# B&R Automation Studio project 8238 (part 29)

#### BIN_TO_BCD_INT.ab
```automation-basic
FUNCTION_BLOCK BIN_TO_BCD_INT

		(* Implementation of BIN_TO_BCD *)

	RegisterOUT = 0

		remain = RegisterIN

;		f = remain / 100000
;		remain = remain - (f * 100000)
;		e = remain / 10000
;		remain = remain - (e * 10000)
		d = remain / 1000
		remain = remain - (d * 1000)
		c = remain / 100
		remain = remain - (c * 100)
		b = remain / 10
		a = remain - (b * 10)
		RegisterOUT = RegisterIN + (b * 6) + (c * 156) + (d * 3096)// + (e * 55536)// + (f * 948576)

END_FUNCTION_BLOCK
```

#### Get_Lower2Bytes.st
```iecst
(* Copy the lower 2 bytes from a byte register *)
FUNCTION Get_Lower2Bytes

	memcpy(ADR(Get_Lower2Bytes),ADR(input),2);

END_FUNCTION
```

#### Get_Higher2Bytes.st
```iecst
(* Copy the upper 2 bytes of a DWORD to a WORD *)
FUNCTION Get_Higher2Bytes
	memcpy(ADR(Get_Higher2Bytes),ADR(input) + 2,2);
END_FUNCTION
```

#### GetPowerlinkNodeIP.st
```iecst
(* *Function to build BR camera image URL from EPL IP and Node address *)
FUNCTION_BLOCK GetPowerlinkNodeIP

	IF EDGEPOS(Enable)AND (state = 0) THEN
		state := 1;
	ELSIF (((state = 4) OR (state = 100)) AND NOT Enable) THEN
		state := 0;
	END_IF;

	getEPL_IP.enable 	:= (state = 2);

	CASE state OF
		0:  // WAIT
			Status := ERR_FUB_ENABLE_FALSE;

		1: // Build and check the interface path
			Status := ERR_FUB_BUSY;
			IF (RIGHT(EplInterfacePath,4) = '.ETH') THEN
				device := EplInterfacePath;
				state := 2;
			ELSE
				device := CONCAT(EplInterfacePath,'.ETH');
				state := 2;
			END_IF;

		2:// Get the IP address of the interface..
			Status := ERR_FUB_BUSY;
			getEPL_IP.pIPAddr 	:= ADR(eplAddress);
			getEPL_IP.Len 		:= SIZEOF(eplAddress);
			getEPL_IP.pDevice 	:= ADR(device);
			IF (getEPL_IP.status = ERR_OK) THEN
				state := 3;
				//brsstrcpy(pIPAddress,ADR(''));
			ELSIF (getEPL_IP.status <> ERR_FUB_BUSY) AND (getEPL_IP.status <> ERR_FUB_ENABLE_FALSE)  THEN
				Status := getEPL_IP.status;
				state := 100;
			END_IF;

		3://Replace the
			Status := ERR_FUB_BUSY;
			ethInetAton(ADR(eplAddress),ADR(eplIP));
			eplIP := (eplIP AND 16#00FF_FFFF) OR (16#FF00_0000 AND SHL(Node,24));// Replace the end of the IP with the node
			ethInetNtoa(eplIP,pIPAddress);
			state := 4;

		4:// Complete
			Status := ERR_OK;

		100:// Error step

	END_CASE;

	getEPL_IP();

END_FUNCTION_BLOCK
```

#### DByte_TO_4Byte.st
```iecst
(* Build 32 bit register from 2 16bit register *)
FUNCTION DByte_TO_4Byte
	memcpy(ADR(internalValue),adrLower,2);
	memcpy(ADR(internalValue)+2,adrHigher,2);
	DByte_TO_4Byte := internalValue;
END_FUNCTION
```

#### getNodeFromPV.st
```iecst
(* Get Node and Connection string from a PV var. *)
FUNCTION_BLOCK getNodeFromPV

	IF NOT enable THEN
		state := 0;
	END_IF;

	IF (state = 0) THEN // Not ENABLED
		IF enable THEN
			state := 1;
			pointer := 0;
			IF_Adr := '';
			NodeNumber := 0;
			brsmemset(ADR(searchString),0,SIZEOF(searchString));
		ELSE
			status := ERR_FUB_ENABLE_FALSE;
		END_IF;
	END_IF;

	IF (state = 1) THEN // get pointer to iom file so we can interate through the string.
		searchLen := LEN(pvName);
		mO_info(enable := (searchLen > 0), pName := ADR('iomap'), grp := 0);
		IF ((searchLen = 0) OR (searchLen > SIZEOF(searchString))) THEN
			state := 100;
			status := 101;
		ELSIF (mO_info.status = ERR_OK) THEN
			state := state := 2;
		ELSIF (mO_info.status <> ERR_FUB_BUSY) THEN
			status := mO_info.status;
			state := 100;
		END_IF;
	END_IF;

	//iterate through the string until we find our var name
	scanCount := 0;
	WHILE ((pointer < (mO_info.size - searchLen)) AND (scanCount <= 50000) AND (state = 2)) DO
		scanCount := scanCount + 1;
		brsmemcpy(ADR(searchString),(mO_info.address + pointer),searchLen);
		IF (searchString = pvName) THEN
			brsmemset(ADR(searchString),0,SIZEOF(searchString));
			state := 3;
		END_IF;
		pointer := pointer + 1;
		IF (pointer = (mO_info.size - searchLen)) THEN
			state := 20; // NOT FOUND
		END_IF;
	END_WHILE;

	// Iterate back through the string to find the start of the node
	scanCount := 0;
	WHILE ((pointer > 0) AND (pointer < (mO_info.size - searchLen)) AND (scanCount <= 250) AND (state = 3)) DO
		scanCount := scanCount + 1;
		pointer := pointer - 1;
		brsmemcpy(ADR(searchString),(mO_info.address + pointer),2);
		IF (searchString = 'ST') THEN
			startNode := pointer + 2;
			brsmemset(ADR(searchString),0,SIZEOF(searchString));
			state := 4;
		END_IF;
		IF (pointer = 0) OR (scanCount = 250) THEN
			state := 100; // ERROR;
			status := 103;
		END_IF;
	END_WHILE;

	// Iterate back through the string to find the start of the path
	scanCount := 0;
	WHILE ((pointer > 0) AND (pointer < (mO_info.size - searchLen)) AND (scanCount <= 250) AND (state = 4)) DO
		scanCount := scanCount + 1;
		pointer := pointer - 1;
		brsmemcpy(ADR(searchString),(mO_info.address + pointer),2);
		IF (searchString = '="') THEN
			startPath := pointer + 2;
			pointer := startNode;
			brsmemset(ADR(searchString),0,SIZEOF(searchString));
			state := 5;
		END_IF;
		IF (pointer = 0) OR (scanCount = 250) THEN
			state := 100; // ERROR;
			status := 104;
		END_IF;
	END_WHILE;

	// Iterate back through the string to find the end of the node
	scanCount := 0;
	WHILE ((pointer > 0) AND (pointer < (mO_info.size - 1)) AND (scanCount <= 250) AND (state = 5)) DO
		scanCount := scanCount + 1;
		pointer := pointer + 1;
		brsmemcpy(ADR(searchString),(mO_info.address + pointer),1);
		IF (searchString = '"') OR (searchString = '.') THEN
			endNode := pointer;
			state := 6;
		END_IF;
		IF (pointer = 0) OR (pointer = (mO_info.size - 1)) OR (scanCount = 250) THEN
			state := 100; // ERROR;
			status := 105;
		END_IF;
	END_WHILE;

	IF (state = 6) THEN
		brsmemset(ADR(IF_Adr),0,SIZEOF(IF_Adr));
		brsmemcpy(ADR(IF_Adr),mO_info.address + startPath, startNode - 3 - startPath);
		IF (LEFT(IF_Adr,1) = '%') THEN
			 IF_Adr := RIGHT(IF_Adr,(LEN(IF_Adr) - 4));
		END_IF;
		// Get the Node
		brsmemset(ADR(nodeString),0,SIZEOF(nodeString));
		brsmemcpy(ADR(nodeString),mO_info.address + startNode, endNode - startNode);
		NodeNumber := DINT_TO_USINT(atoi(ADR(nodeString)));
		state := 10;
	END_IF;

	IF (state = 10) THEN// Complete

	END_IF;

	IF (state = 20) THEN // NOT FOUND

	END_IF;

	IF (state = 100) THEN // ERROR
		state := 0;
	END_IF;

	IF (state = 10) THEN
		status := ERR_OK;
		state := 0;
	ELSIF (state = 20) THEN // NOT FOUND
		status := 200; // NOT FOUND
		state := 0;
	ELSIF (state > 0) AND (state < 100) THEN
		status := ERR_FUB_BUSY;
	END_IF;

END_FUNCTION_BLOCK
```

#### GetModuleName.st
```iecst
(* TODO: Add your comment here *)
FUNCTION_BLOCK GetModuleName

	IF NOT enable THEN
		state := 0;
	END_IF;

	IF (state = 0) THEN // Not ENABLED
		IF enable THEN
			state := 1;
			pointer := 0;
		ELSE
			status := ERR_FUB_ENABLE_FALSE;
		END_IF;
	END_IF;

	IF (state = 1) THEN // get pointer to iom file so we can interate through the string.
		brsstrcpy(ADR(moduleAddress),ADR('"'));
		brsstrcat(ADR(moduleAddress),pModuleAddress);
		brsstrcat(ADR(moduleAddress),ADR('"'));
		brsmemset(ADR(searchString),0,SIZEOF(searchString));
		brsmemset(ADR(ModuleName),0,SIZEOF(ModuleName));
		searchLen := LEN(moduleAddress);
		mO_info(enable := (searchLen > 0), pName := ADR('arconfig'), grp := 0);
		IF ((searchLen <= 2) OR (searchLen > SIZEOF(searchString))) THEN
			state := 100;
			status := 101;
		ELSIF (mO_info.status = ERR_OK) THEN
			state := state := 2;
		ELSIF (mO_info.status <> ERR_FUB_BUSY) THEN
			status := mO_info.status;
			state := 100;
		END_IF;
	END_IF;

	//iterate through the string until we find our address
	scanCount := 0;
	WHILE ((pointer < (mO_info.size - searchLen)) AND (scanCount <= 50000) AND (state = 2)) DO
		scanCount := scanCount + 1;
		brsmemcpy(ADR(searchString),(mO_info.address + pointer),searchLen);
		IF (searchString = moduleAddress) THEN
			brsmemset(ADR(searchString),0,SIZEOF(searchString));
			foundCount := foundCount + 1;
			state := 3;
		END_IF;
		pointer := pointer + 1;
		IF (pointer = (mO_info.size - searchLen)) THEN
			state := 20; // NOT FOUND
		END_IF;
	END_WHILE;

	// Iterate back through the string to find the module Name
	scanCount := 0;
	WHILE ((pointer > 0) AND (pointer < (mO_info.size - 1)) AND (scanCount <= 200) AND (state = 3)) DO
		scanCount := scanCount + 1;
		pointer := pointer + 1;
		brsmemcpy(ADR(searchString),(mO_info.address + pointer),42);
		IF (searchString = '<Parameter ID="HardwareModuleName" Value="')THEN
			brsmemset(ADR(searchString),0,SIZEOF(searchString));
			pointer := pointer + 42;
			start := pointer;
			state := 4;
		END_IF;
		IF (pointer = 0) OR (pointer = (mO_info.size - 1)) OR (scanCount = 200) THEN
			state := 100; // ERROR;
			status := 103;
		END_IF;
	END_WHILE;

	// Iterate back through the string to find the module Name
	scanCount := 0;
	WHILE ((pointer > 0) AND (pointer < (mO_info.size - 1)) AND (scanCount <= 100) AND (state = 4)) DO
		scanCount := scanCount + 1;
		pointer := pointer + 1;
		brsmemcpy(ADR(searchString),(mO_info.address + pointer),1);
		IF (searchString = '"')THEN
			end := pointer;
			state := 5;
		END_IF;
		IF (pointer = 0) OR (pointer = (mO_info.size - 1)) OR (scanCount = 100) THEN
			state := 100; // ERROR;
			status := 104;
		END_IF;
	END_WHILE;

	IF (state = 5) THEN
		// Get the Name
		IF ((end - start) <= SIZEOF(ModuleName)) THEN
			brsmemset(ADR(ModuleName),0,SIZEOF(ModuleName));
			brsmemcpy(ADR(ModuleName),mO_info.address + start, end - start);
			state := 10;
		ELSE
			state := 100;
			status := 105;
		END_IF;
	END_IF;

	IF (state = 10) THEN// Complete

	END_IF;

	IF (state = 20) THEN // NOT FOUND

	END_IF;

	IF (state = 100) THEN // ERROR
		state := 0;
	END_IF;

	IF (state = 10) THEN
		status := ERR_OK;
		state := 0;
	ELSIF (state = 20) THEN // NOT FOUND
		status := 200; // NOT FOUND
		state := 0;
	ELSIF (state > 0) AND (state < 100) THEN
		status := ERR_FUB_BUSY;
	END_IF;

END_FUNCTION_BLOCK
```

#### Get_LowerByte.st
```iecst
(* Copy the lower 2 bytes from a byte register *)
FUNCTION Get_LowerByte

	memcpy(ADR(Get_LowerByte),ADR(input),1);

END_FUNCTION
```

#### Get_HigherByte.st
```iecst
(* Copy the upper 2 bytes of a DWORD to a WORD *)
FUNCTION Get_HigherByte
	memcpy(ADR(Get_HigherByte),ADR(input) + 1,1);
END_FUNCTION
```

#### SetValueByName.st
```iecst
//*Set Local variable from external task
FUNCTION SetValueByName
	SetValueByName := 0;
	IF (brsstrlen(ADR(TaskName)) > 0 )THEN
		varName := '::';
		brsstrcat(ADR(varName),ADR(TaskName));
		brsstrcat(ADR(varName),ADR(':'));
		brsstrcat(ADR(varName),ADR(VarName));
	ELSE
		brsstrcpy(ADR(varName),ADR(VarName));
	END_IF;

	IF (PV_xgetadr(ADR(varName),ADR(pVar),ADR(sVar)) = 0) THEN
		IF (SIZEOF(Value) <= sVar)THEN
			brsmemcpy(pVar,ADR(Value),SIZEOF(Value));
			SetValueByName := 1;
		ELSE
			brsmemcpy(pVar,ADR(Value),sVar);
			SetValueByName := 1;
		END_IF;
	END_IF;
END_FUNCTION
```

#### GetValueByName.st
```iecst
//*Set Local variable from external task
FUNCTION GetValueByName
	GetValueByName := 0;

	IF (brsstrlen(ADR(TaskName)) > 0 )THEN
		varName := '::';
		brsstrcat(ADR(varName),ADR(TaskName));
		brsstrcat(ADR(varName),ADR(':'));
		brsstrcat(ADR(varName),ADR(VarName));
	ELSE
		brsstrcpy(ADR(varName),ADR(VarName));
	END_IF;

	status := PV_xgetadr(ADR(varName),ADR(pVar),ADR(sVar));
	IF (status = 0) THEN
		IF (sValue >= sVar)THEN
			//Clear the value
			IF (sValue > sVar) THEN
				brsmemset(pValue,0,sValue);
			END_IF;
			brsmemcpy(pValue,pVar,sVar);
			GetValueByName := 1;
		END_IF;
	END_IF;
END_FUNCTION
```

#### LoadCell.st
```iecst
FUNCTION_BLOCK LoadCell

	IF capture_weight_bool THEN
		brsmemmove(ADR(weight_array[1]), ADR(weight_array), 1498);

		weight_array[0] := analog_weight;

		IF small_interval > 0 THEN
			small_value := 0;
			FOR i := 0 TO small_interval - 1 DO
			small_value := small_value + weight_array[i];
			END_FOR;
			udp_data.small_smoothing_value := small_smoothing_value := DINT_TO_UINT(small_value / small_interval);

		END_IF;

		IF large_interval > 0 THEN
			large_value := 0;
			FOR x := 0 TO large_interval - 1 DO
			large_value := large_value + weight_array[x];
			END_FOR;

			udp_data.large_smoothing_value := large_smoothing_value := DINT_TO_UINT(large_value / large_interval);
		END_IF;

		udp_data.capture_weight := capture_weight := analog_weight;
	END_IF;

	weight_tolerance := (((server_send_weight - tare)/100) * weight_tolerance_percent);
	empty := (analog_weight <= (tare + weight_tolerance)) AND (tare > 0);
	min_weight:= (analog_weight > server_min_weight) AND (server_min_weight > 0);
	near_weight := (analog_weight > server_near_weight) AND (server_near_weight > 0);
	bufflector_door_weight := (analog_weight > server_buffer_weight) AND (server_buffer_weight > 0);
	notify_weight := (analog_weight > server_notify_weight) AND (server_notify_weight > 0);
	full := (analog_weight > server_send_weight) AND (server_send_weight > 0);
	over_weight:= (analog_weight >= server_over_weight);

	IF span > 0 THEN
		udp_data.capture_weight_value := capture_weight_value := (((udp_data.capture_weight - tare) * 100) / span);
		udp_data.live_weight_value := live_weight_value := (((analog_weight - tare) * 100) / span);
		udp_data.small_smoothing_weight := small_smoothing_weight := (((udp_data.small_smoothing_value - tare) * 100) / span);
		udp_data.large_smoothing_weight := large_smoothing_weight := (((udp_data.large_smoothing_value - tare) * 100) / span);
	END_IF;

END_FUNCTION_BLOCK
```

#### BCD_ENCODE.st
```iecst
(* TODO: Add your comment here *)
FUNCTION_BLOCK BCD_Encode

	Output := 0;

	IF Input.0 THEN
		Output := Output + 1;
	END_IF;
	IF Input.1 THEN
		Output := Output + 2;
	END_IF;
	IF Input.2 THEN
		Output := Output + 4;
	END_IF;
	IF Input.3 THEN
		Output := Output + 8;
	END_IF;
	IF Input.4 THEN
		Output := Output + 10;
	END_IF;
	IF Input.5 THEN
		Output := Output + 20;
	END_IF;
	IF Input.6 THEN
		Output := Output + 40;
	END_IF;
	IF Input.7 THEN
		Output := Output + 80;
	END_IF;
	IF Input.8 THEN
		Output := Output + 100;
	END_IF;
	IF Input.9 THEN
		Output := Output + 200;
	END_IF;
	IF Input.10 THEN
		Output := Output + 400;
	END_IF;
	IF Input.11 THEN
		Output := Output + 800;
	END_IF;
	IF Input.12 THEN
		Output := Output + 1000;
	END_IF;
	IF Input.13 THEN
		Output := Output + 2000;
	END_IF;
	IF Input.14 THEN
		Output := Output + 4000;
	END_IF;
	IF Input.15 THEN
		Output := Output + 8000;
	END_IF;

END_FUNCTION_BLOCK
```

#### Types.typ
```iecst
TYPE
RailComm_typ :STRUCT
  Messages : RailMessages_typ;
END_STRUCT;
RailMessages_typ : STRUCT
  Write : UINT;
  Read : ARRAY[0..15] OF UINT;
END_STRUCT;
SlingInput_typ : STRUCT
  Write : UINT;
  Read : UDINT;
END_STRUCT;
  bnr_io : STRUCT
    X01 : BOOL;
    X02 : BOOL;
    X03 : BOOL;
    X04 : BOOL;
    X05 : BOOL;
    X06 : BOOL;
    X07 : BOOL;
    X08 : BOOL;
    X09 : BOOL;
    X10 : BOOL;
    X11 : BOOL;
    X12 : BOOL;
    X13 : BOOL;
    X14 : BOOL;
    X15 : BOOL;
    X16 : BOOL;
    X17 : BOOL;
    X18 : BOOL;
    X19 : BOOL;
    X20 : BOOL;
    Y01 : BOOL;
    Y02 : BOOL;
    Y03 : BOOL;
    Y04 : BOOL;
    Y05 : BOOL;
    Y06 : BOOL;
    Y07 : BOOL;
    Y08 : BOOL;
    Y09 : BOOL;
    Y10 : BOOL;
    Y11 : BOOL;
    Y12 : BOOL;
    Y13 : BOOL;
    Y14 : BOOL;
    Y15 : BOOL;
    Y16 : BOOL;
    Y17 : BOOL;
    Y18 : BOOL;
    Y19 : BOOL;
    Y20 : BOOL;
  END_STRUCT;

  rail : 	STRUCT
    ac : BOOL;
    activity : BOOL;
    after : BOOL;
    after_raw : BOOL;
    after_a : BOOL;
    after_a_raw : BOOL;
    after_b : BOOL;
    after_b_raw : BOOL;
    air_pressure : BOOL;
    alarm : BOOL;
    alarm_time : TIME;
    arm: BOOL;
    arrive : BOOL;
    arrive_raw : BOOL;
    at_rail : BOOL;
    bag_emptied : BOOL;
    before : BOOL;
    before_raw : BOOL;
    bnx : BOOL;
    bottom_door : BOOL;
    bottom_door_sensor : BOOL;
    bring_ok : BOOL;
    bufflector_door_weight : BOOL;
    buffer_protection : BOOL;
    busy : BOOL;
    cake_break_bypass : BOOL;
    cake_break_done : BOOL;
    cake_break_signal : BOOL;
    cake_break_start : BOOL;
    cake_close : BOOL;
    cake_left : BOOL;
    cake_open : BOOL;
    cake_right : BOOL;
    call_button : BOOL;
    capture_weight: BOOL;
    catch : BOOL;
    cc_open_bottom : BOOL;
    cc_open_bottom_os : BOOL;
    cc_open_top : BOOL;
    cc_open_top_os : BOOL;
    cc_shut_bottom : BOOL;
    cc_shut_bottom_os : BOOL;
    cc_shut_top : BOOL;
    cc_shut_top_os : BOOL;
    change_reset : BOOL;
    chute : BOOL;
    chute_clear : BOOL;
    chute_in_position : BOOL;
    clamp : BOOL;
    clear_belt : BOOL;
    close : BOOL;
    close_bottom : BOOL;
    close_top : BOOL;
    closed : BOOL;
    comm_ok : BOOL;
    counter : USINT;
    conv_estop : BOOL;
    conv_fwd : BOOL;
    conv_rev : BOOL;
    conveyor_running : BOOL;
    custom_bring_lock : BOOL;
    custom_send_lock : BOOL;
    cycle_count : INT;
    cylinderAtReceive : BOOL;
    cylinderAtRelease : BOOL;
    dampner : BOOL;
    dampner_closed : BOOL;
    dampner_open : BOOL;
    debagger_arm : BOOL;
    delayed_bottom_door : BOOL;
    destination : INT;
    device_received : BOOL;
    device_receive_ok : BOOL;
    device_release_ok : BOOL;
    dog_sensor : BOOL;
    done : BOOL;
    done_smashing : BOOL;
    door_sensor : BOOL;
    down : BOOL;
    down_button : BOOL;
    down_raw : BOOL;
    emergency_cut_off : BOOL;
    empty : BOOL;
    empty_bag : BOOL;
    energize : BOOL;
    fire : BOOL;
    fire_cyl_receive : BOOL;
    fire_cyl_release : BOOL;
    fire_down : BOOL;
    fire_f_trig : F_TRIG;
    fire_r_trig : R_TRIG;
    fire_ns : BOOL;
    fire_os : BOOL;
    fire_up : BOOL;
    fired: BOOL;
    firing : BOOL;
    firing_reset : BOOL;
    flip : BOOL;
    flipped : BOOL;
    fnx : BOOL;
    foot : BOOL;
    front : BOOL;
    front_a : BOOL;
    front_b : BOOL;
    front_bag_mt : BOOL;
    front_raw : BOOL;
    front_stp : BOOL;
    full : BOOL;
    full_sensor : BOOL;
    green_light : BOOL;
    going_to : BOOL;
    going_to_os : BOOL;
    going_to_ns : BOOL;
    going_to_r_trig : R_TRIG;
    going_to_f_trig : F_TRIG;
    grab : BOOL;
    high_valve : BOOL;
    input_enabled : BOOL;
    insert : BOOL;
    insert_reset : BOOL;
    in_pos : BOOL; (*In position after dbnc*)
    in_pos_raw : BOOL;  (*In position sensor*)
    inx : BOOL;
    io_ok : BOOL;
    io_ok_A : BOOL;
    io_ok_B : BOOL;
    io_ok_C : BOOL;
    jogmode : BOOL;
    latch : BOOL;
    latched : BOOL;
    leave1 : BOOL;
    leave2 : BOOL;
    leave3 : BOOL;
    level_arm : BOOL;
    lift_stp : BOOL;
    LFT1 : BOOL;
    LFT1_RAW : BOOL;
    LFT2 : BOOL;
    LFT2_RAW : BOOL;
    LFT3 : BOOL;
    LFT3_RAW : BOOL;
    LFT4 : BOOL;
    LFT4_RAW : BOOL;
    LFT5 : BOOL;
    LFT5_RAW : BOOL;
    lift_clamp : BOOL;
    lift_jammed : BOOL;
    lift_position : INT;
    lift_running : BOOL;
    loaded : BOOL;
    loading_position : BOOL;
    loading_position_raw : BOOL;
    loading_signal : BOOL;
    lockout : BOOL;
    log_dist : INT;
    log_now_a : BOOL;
    log_now_b : BOOL;
    low_air_alarm : BOOL;
    low_valve : BOOL;
    man_open : BOOL;
    man_send : BOOL;
    man_send_button_1 : BOOL;
    man_send_button_2 : BOOL;
    man_send_button : BOOL;
    manual_mode : BOOL;
    marker_made : BOOL;
    mid : BOOL;
    mid_raw : BOOL;
    min_weight : BOOL;
    min_weight_send : BOOL;
    mod_count : INT;
    move_rail : BOOL;
    move_rail_up : BOOL;
    move_rail_down : BOOL;
    mt_arrived : BOOL;
    near_weight : BOOL;
    near_weight_send : BOOL;
    need_to_empty_bd : BOOL;
    need_to_empty_td : BOOL;
    next_rails_ok : BOOL;
    no_dests_ok : BOOL;
    not_io_ok : BOOL;
    notify_weight : BOOL;
    oc : BOOL;
    ok_to_send : BOOL;
    onoff : BOOL;
    open : BOOL;
    open_bottom : BOOL;
    open_manual : BOOL;
    open_signal : BOOL;
    open_pendant : BOOL;
    opened : BOOL;
    out1 : BOOL;
    over_full_sensor : BOOL;
    over_full_light : BOOL;
    over_weight : BOOL;
    paddle_sensor : BOOL;
    pilot_light : BOOL;
    poa : BOOL;
    pos1 : BOOL;
    pos1_raw : BOOL;
    pos2 : BOOL;
    pos2_raw : BOOL;
    pos3 : BOOL;
    pos3_raw : BOOL;
    pos4 : BOOL;
    pos4_raw : BOOL;
    pos_1_after_raw : BOOL;
    pos_1_after : BOOL;
    pos_2_after_raw : BOOL;
    pos_2_after : BOOL;
    pos_3_after_raw : BOOL;
    pos_3_after : BOOL;
    pos_4_after_raw : BOOL;
    pos_4_after : BOOL;
    pos_5_after_raw : BOOL;
    pos_5_after : BOOL;
    pos_6_after_raw : BOOL;
    pos_6_after : BOOL;
    preceeding_rails_ok : BOOL;
    pressure_full_line_1 : BOOL;
    pressure_full_line_2 : BOOL;
    pressure_full_line_3 : BOOL;
    pressure_sensor : BOOL;
    pressure_sensor_1 : BOOL;
    pressure_sensor_2 : BOOL;
    pressure_sensor_3 : BOOL;
    pressure_stop : BOOL;
    pressure_stop_1 : BOOL;
    pressure_stop_2 : BOOL;
    pressure_stop_3 : BOOL;
    prox1 : BOOL;
    prox1_raw : BOOL;
    prox2 : BOOL;
    prox2_raw : BOOL;
    prs_a : BOOL;
    prs_b : BOOL;
    prs_1 : BOOL;
    prs_2 : BOOL;
    prs_3 : BOOL;
    prs_4 : BOOL;
    prs_5 : BOOL;
    prs_6 : BOOL;
    purge : BOOL;
    pusher : BOOL;
    puncher : BOOL;
    ratchet: BOOL;
    rail_full : BOOL;
    rail_mt : BOOL;
    rail_out_sensor : BOOL;
    rail_sensor: BOOL;
    raise_to_send : BOOL;
    ratchet_position : INT := 0;
    ready_to_send : BOOL;
    rear : BOOL;
    rear_raw : BOOL;
    rear_stp : BOOL;
    receive_manual : BOOL;
    receive_signal : BOOL;
    receive_pendant : BOOL;
    receive_position : BOOL;
    receive_position_raw : BOOL;
    received : BOOL;
    receiving : BOOL;
    red_light : BOOL;
    release_position : BOOL;
    release_position_raw : BOOL;
    releasing : BOOL;
    remove : BOOL;
    remove_reset : BOOL;
    reset : BOOL;
    reset_switch : BOOL;
    retry : BOOL;
    request_rotate: BOOL; (* Bit for Supertrack rotaty point types - so the plc knows to rotate. *)
    ring_pusher : BOOL;
    run_conveyor : BOOL;
    run_slant : BOOL;
    running : BOOL;
    safety : BOOL;
    safety_zone : BOOL;
    safety_stop : BOOL;
    safety_stop_1 : BOOL;
    safety_stop_2 : BOOL;
    safety_stop_3 : BOOL;
    safety_stop_4 : BOOL;
    safety_stop_5 : BOOL;
    safety_stop_6 : BOOL;
    send_button : BOOL;
    send_manual : BOOL;
    send_ok : BOOL;
    send_ready : BOOL;
    sending : BOOL;
    sent : BOOL;
    servo_command : INT;
    servo_position : INT;
    slant_inx : BOOL;
    sort_entry_clear : BOOL;
    sort_exit_clear : BOOL;
    short_stroke : BOOL;
    shut : BOOL;
    simple_lockout : BOOL;
    sis_weight_not_ok : BOOL;
    sis_weight_ok : BOOL;
    sling_ready : BOOL;
    smashed1 : BOOL;
    smashed2 : BOOL;
    state : INT;
    static_close : BOOL;
    static_open : BOOL;
    stb : BOOL;
    stb_delay : BOOL;
    stb_down : BOOL;
    stb_up : BOOL;
    start_button : BOOL;
    stop_button : BOOL;
    stopped : BOOL;
    stp : BOOL;
    stp_a : BOOL;
    stp_b : BOOL;
    sw_in_a : BOOL;
    sw_in_b : BOOL;
    sw_out_a : BOOL;
    sw_out_b : BOOL;
    swa : BOOL;
    swb : BOOL;
    swc : BOOL;
    switch : BOOL;
    switch_delay : BOOL;
    switch_trigger : BOOL;
    swx : BOOL;
    swy : BOOL;
    swz : BOOL;
    table_up : BOOL;
    table_down : BOOL;
    tilt_arm : BOOL;
    timeout : BOOL;
    to_pos1 : BOOL;
    to_pos2 : BOOL;
    to_pos3 : BOOL;
    to_pos4 : BOOL;
    top_door : BOOL;
    top_door_lock : BOOL;
    top_door_delay : BOOL;
    top_rail_busy : BOOL;
    transfer_requested_signal : BOOL;
    trolley_seen : BOOL;
    trolley_seen_delay : BOOL;
    up : BOOL;
    up_button : BOOL;
    up_raw : BOOL;
    upper_down : BOOL;
    upper_up : BOOL;
    wait_for_mt : BOOL;
    wait_for_mt_bd : BOOL;
    wait_for_mt_td : BOOL;
    waiting : BOOL;
    weight_ok : BOOL;
    xfer_complete : BOOL;
    xfer_in_progress : BOOL;
    want_to_run : BOOL;
    warning : BOOL;
    warning_com : INT;
    zone_clear : BOOL;
  END_STRUCT;

  SinglePanelStatusArray : STRUCT
    panels : ARRAY[0..3] OF INT;
  END_STRUCT;

  BC : STRUCT
    VDC_OK : BOOL;
  END_STRUCT;

  Weight_typ : STRUCT
    Wgt_Channel_1 : DINT;
    Wgt_Channel_2 : DINT;
    Config_Channel_1 : USINT;
    Config_Channel_2 : USINT;
  END_STRUCT;

  CakeBreaker : STRUCT
    both_clear : BOOL;
    both_seen : BOOL;
    cake_close : BOOL;
    cake_left : BOOL;
    cake_open : BOOL;
    cake_right : BOOL;
    crushes_after_seen : INT := 3;
    crushes_before_check : INT := 3;
    crush_count : INT := 0;
    done : BOOL;
    flutter_count : INT := 0;
    reset : BOOL;
    seen_count : INT := 0;
    sling_loading_flutters : INT := 5;
    start : BOOL;
    state : INT := 0;
    total_crushes : INT := 20;
    CrushCloseTimer : TON;
    CrushCloseTime : INT := 5000;
    CrushOpenTimer : TON;
    CrushOpenTime : INT := 3000;
    HalfCrushCloseTimer : TON;
    HalfCrushCloseTime : INT := 2500;
    HalfCrushOpenTimer : TON;
    HalfCrushOpenTime : INT := 1500;
    FlutterCloseTimer : TON;
    FlutterCloseTime : INT := 750;
    FlutterOpenTimer : TON;
    FlutterOpenTime : INT := 1000;
  END_STRUCT;

   LoadcellUdpType : STRUCT
     capture_weight : UINT;
     capture_weight_value : UINT;
     small_smoothing_value : UINT;
     large_smoothing_value :UINT;
     large_smoothing_weight : UINT;
     live_weight_value : UINT;
     small_smoothing_weight : UINT;
   END_STRUCT;

  RailUdpType : STRUCT
    state : INT;
    waiting : BOOL;
    bring_ok : BOOL;
    alarm : BOOL;
    warning_com : INT;
  END_STRUCT;

END_TYPE
```

#### SupertrackIndexerUnTracked.st
```iecst
(* TODO: Add your comment here *)
FUNCTION_BLOCK SupertrackIndexerUnTracked

	messages ACCESS p_messages;

	  // Debounce Inputs
	DBNC_front_timer(IN := front_raw, PT := DBNC_front_time);
	front := DBNC_front_timer.Q;

	DBNC_arrive_timer(IN := arrive_raw, PT := DBNC_arrive_time);
	arrive := DBNC_arrive_timer.Q;

	DBNC_after_timer(IN := after_raw, PT := DBNC_after_time);
	after := DBNC_after_timer.Q;

	// Device State Machine
	IF reset THEN udp_data.state := state := ReadyToRelease; END_IF;
	IF udp_data.state = 0 THEN udp_data.state := state := ReadyToRelease; END_IF;

	CASE udp_data.state OF
		ReadyToRelease:
			IF fire_os THEN
				udp_data.state := state := Releasing;
			END_IF;

		Releasing:
			IF after OR NOT(fire) THEN
				udp_data.state := state := ReadyToRelease;
			END_IF;

	END_CASE;

	// Comm Logic
	udp_data.waiting := waiting := (
	udp_data.state = ReadyToRelease
	AND front
	AND NOT(custom_send_lock)
	AND NOT(after)
	AND NOT(safety_zone)
	);

	udp_data.bring_ok := bring_ok := (
	NOT(before)
	AND NOT(arrive)
	AND NOT(going_to)
	AND NOT(custom_bring_lock)
	AND (counter = 2)
	);

	IF going_to AND arrive THEN insert := TRUE; END_IF;

	// Trolley Counting
	IF reset THEN
		counter := 2;
	END_IF;

	IF EDGEPOS(going_to) THEN
		counter := 0;
	END_IF;

	IF EDGEPOS(arrive_raw) AND NOT(INS_OFF.Q) THEN
		IF (counter < 2 )THEN
			counter := counter + 1;
		END_IF;
	END_IF;

	IF ok_to_send THEN
		IF rail_full THEN
			counter := 1;
		ELSE
			counter := 2;
		END_IF;
		ok_to_send := 0;
	END_IF;

	INS_OFF(IN := (arrive_raw), PT := DBNC_counter_time);

	// Output Control
	inx := udp_data.state = Releasing;

	// Pressure Relief
	tof_pressure(IN := pressure_full_line_1, PT:= tof_pressureTime);
	pressure_stop_1 := NOT tof_pressure.Q;

	tof_pressure_2(IN := pressure_full_line_2, PT:= tof_pressureTime);
	pressure_stop_2 := NOT tof_pressure_2.Q;

	tof_pressure_3(IN := pressure_full_line_3, PT:= tof_pressureTime);
	pressure_stop_3 := NOT tof_pressure_3.Q;

	tof_pressure_4(IN := pressure_full_line_4, PT:= tof_pressureTime);
	pressure_stop_4 := NOT tof_pressure_4.Q;

	tof_pressure_5(IN := pressure_full_line_5, PT:= tof_pressureTime);
	pressure_stop_5 := NOT tof_pressure_5.Q;

	// Alarm Timers
	AlarmTimer(IN := fire, PT := (t#1s * rail_alarm_time));
	UnexpectedBagTimer(IN := (arrive AND NOT(front) AND NOT(inx)), PT := UnexpectedBagTime);
	RearTrolleyLockTimer(IN := (counter = 0) AND NOT(front) AND NOT(going_to), PT := RearTrolleyLockTime);

	// Alarm Coms
	udp_data.alarm := alarm := AlarmTimer.Q;
	udp_data.warning_com.0 := warning_com.0 := UnexpectedBagTimer.Q;
	udp_data.warning_com.2 := warning_com.2 := RearTrolleyLockTimer.Q;

	messages.Write := 0;
	IF UnexpectedBagTimer.Q   THEN messages.Write := BIT_SET(messages.Write,UNEXPECTED_BAG); END_IF;
	IF RearTrolleyLockTimer.Q      THEN messages.Write := BIT_SET(messages.Write,REAR_TROLLEY_LOCK); END_IF;

	// Always clear acknowledgements
	brsmemset(ADR(messages.Read[0]),0,SIZEOF(messages.Read));

END_FUNCTION_BLOCK
```

#### SupertrackIndexerTracked.st
```iecst
(* TODO: Add your comment here *)
FUNCTION_BLOCK SupertrackIndexerTracked

	messages ACCESS p_messages;

	  // Debounce Inputs
	DBNC_front_timer(IN := front_raw, PT := DBNC_front_time);
	front := DBNC_front_timer.Q;

	DBNC_arrive_timer(IN := arrive_raw, PT := DBNC_arrive_time);
	arrive := DBNC_arrive_timer.Q;

	DBNC_after_timer(IN := after_raw, PT := DBNC_after_time);
	after := DBNC_after_timer.Q;

	// Device State Machine
	IF reset THEN udp_data.state := state := ReadyToRelease; END_IF;
	IF udp_data.state = 0 THEN udp_data.state := state := ReadyToRelease; END_IF;

	CASE udp_data.state OF
		ReadyToRelease:
			IF fire_os THEN
				udp_data.state := state := Releasing;
			END_IF;

		Releasing:
			IF after OR NOT(fire) THEN
				udp_data.state := state := ReadyToRelease;
			END_IF;

	END_CASE;

	// Comm Logic
	udp_data.waiting := waiting := (
	udp_data.state = ReadyToRelease
	AND front
	AND NOT(custom_send_lock)
	AND NOT(after)
	AND NOT(safety_zone)
	AND NOT RearTrolleyLockTimer.IN
	);

	udp_data.bring_ok := bring_ok := (
	NOT(before)
	AND NOT(arrive)
	AND NOT(going_to)
	AND NOT(custom_bring_lock)
	AND (counter = 2)
	);

	IF going_to AND arrive THEN insert := TRUE; END_IF;

	// Trolley Counting
	INS_ON(IN := (rail_mt AND NOT(going_to)), PT := INS_ON_Time);
	IF INS_ON.Q THEN
		counter := 2;
	END_IF;

	IF EDGEPOS(going_to) THEN
		counter := 0;
	END_IF;

	IF EDGEPOS(arrive_raw) AND NOT(INS_OFF.Q) THEN
		IF (counter < 2 )THEN
			counter := counter + 1;
		END_IF;
	END_IF;

	IF ok_to_send THEN
		IF rail_full THEN
			counter := 1;
		ELSE
			counter := 2;
		END_IF;
		ok_to_send := 0;
	END_IF;

	INS_OFF(IN := (arrive_raw), PT := DBNC_counter_time);

	// Output Control
	inx := udp_data.state = Releasing;

	// Pressure Relief
	tof_pressure(IN := pressure_full_line_1, PT:= tof_pressureTime);
	pressure_stop_1 := NOT tof_pressure.Q;

	tof_pressure_2(IN := pressure_full_line_2, PT:= tof_pressureTime);
	pressure_stop_2 := NOT tof_pressure_2.Q;

	tof_pressure_3(IN := pressure_full_line_3, PT:= tof_pressureTime);
	pressure_stop_3 := NOT tof_pressure_3.Q;

	tof_pressure_4(IN := pressure_full_line_4, PT:= tof_pressureTime);
	pressure_stop_4 := NOT tof_pressure_4.Q;

	tof_pressure_5(IN := pressure_full_line_5, PT:= tof_pressureTime);
	pressure_stop_5 := NOT tof_pressure_5.Q;

	// Alarm Timers
	AlarmTimer(IN := fire, PT := (t#1s * rail_alarm_time));
	UnexpectedBagTimer(IN := (front AND rail_mt AND NOT(inx)), PT := UnexpectedBagTime);
	MissingBagTimer(IN := (NOT(front) AND NOT(rail_mt) AND NOT(inx)), PT := MissingBagTime);
	RearTrolleyLockTimer(IN := ((counter = 1) AND NOT rail_full AND NOT inx) OR ((counter = 2) AND rail_full) OR ((counter = 0) AND NOT going_to), PT := RearTrolleyLockTime);

	// Alarm Coms
	udp_data.alarm := alarm := AlarmTimer.Q;
	udp_data.warning_com.0 := warning_com.0 := UnexpectedBagTimer.Q;
	udp_data.warning_com.1 := warning_com.1 := MissingBagTimer.Q;
	udp_data.warning_com.2 := warning_com.2 := RearTrolleyLockTimer.Q;

	messages.Write := 0;
	IF UnexpectedBagTimer.Q   THEN messages.Write := BIT_SET(messages.Write,UNEXPECTED_BAG); END_IF;
	IF MissingBagTimer.Q      THEN messages.Write := BIT_SET(messages.Write,MISSING_BAG); END_IF;
	IF RearTrolleyLockTimer.Q      THEN messages.Write := BIT_SET(messages.Write,REAR_TROLLEY_LOCK); END_IF;

	// Always clear acknowledgements
	brsmemset(ADR(messages.Read[0]),0,SIZEOF(messages.Read));

END_FUNCTION_BLOCK
```

#### SupertrackDischargerStBag.st
```iecst
(* TODO: Add your comment here *)
FUNCTION_BLOCK SupertrackDischargerStBag

	messages ACCESS p_messages;
	loadcell ACCESS p_loadcell;

	// Debounce Inputs
	DBNC_front_timer(IN := front_raw, PT := DBNC_front_time);
	front := DBNC_front_timer.Q;

	DBNC_arrive_timer(IN := arrive_raw, PT := DBNC_arrive_time);
	arrive := DBNC_arrive_timer.Q;

	DBNC_after_timer(IN := after_raw, PT := DBNC_after_time);
	after := DBNC_after_timer.Q;

	// Device State Machine
	IF ResetTimeout.Q THEN
		udp_data.state := state := ReadyToWork;
		man_send := FALSE;
		man_open := FALSE;
	END_IF;
	IF udp_data.state = 0 THEN udp_data.state := state := ReadyToWork; END_IF;

	CASE udp_data.state OF
		ReadyToWork:
			IF NOT(rail_mt) AND front AND onoff AND NOT(halted) AND NOT(ResetTimeout.Q) THEN
				udp_data.state := state := Stabilizing;
			ELSIF man_send THEN
				udp_data.state := state := Destabilizing;
			END_IF;

		Stabilizing:
			static_close := FALSE;
			IF StabilizingTimer.Q THEN
				IF empty_bag OR (messages.Read[BAG_EMPTY_PX] = 1) THEN
					udp_data.state := state := ReadyToTransfer;
				ELSIF (messages.Read[BAG_EMPTY_PX] = 2) THEN
					udp_data.state := state := Destabilizing;
				END_IF;
			ELSIF NOT(onoff) THEN
				udp_data.state := state := ReadyToWork;
			ELSIF man_send THEN
				udp_data.state := state := Destabilizing;
			END_IF;

		ReadyToTransfer:
			IF open_signal OR open_pendant OR man_open THEN
				man_open := FALSE;
				udp_data.state := state := Transferring;
			ELSIF NOT(onoff) THEN
				udp_data.state := state := ReadyToWork;
			ELSIF man_send THEN
				udp_data.state := state := Destabilizing;
				man_send := FALSE;
			END_IF;

		Transferring:
			IF TransferringTimer.Q THEN
				static_close := TRUE;
			END_IF;
			IF receive_signal OR receive_pendant THEN
				udp_data.state := state := LoadReceived;
			ELSIF (messages.Read[TOO_LONG_TO_TRANSFER] > 0) THEN
				CASE messages.Read[TOO_LONG_TO_TRANSFER] OF
					1: //'retry_transfer'
						udp_data.state := state := RetryTransfer;
					2: //'send_bag_away'
						udp_data.state := state := Extending;
				END_CASE;
			ELSIF man_send THEN
				udp_data.state := state := Extending;
				man_send := FALSE;
			END_IF;

		LoadReceived:
			static_close := TRUE;
			IF empty_bag THEN // Bag hasn't opened
				CASE messages.Read[BAG_NOT_OPEN] OF
					1: //'retry_transfer'
						udp_data.state := state := RetryTransfer;
					2: //'send_bag_away'
						udp_data.state := state := Extending;
				END_CASE;
			ELSIF NOT(empty_bag) THEN
				udp_data.state := state := Extending;
			ELSIF man_send THEN
				udp_data.state := state := Extending;
				man_send := FALSE;
			END_IF;

		Extending:
			static_close := TRUE;
			IF ExtendingTimer.Q THEN
				udp_data.state := state := Clamping;
			END_IF;

		Clamping:
			IF ClampingTimer.Q THEN
				udp_data.state := state := Retracting;
			END_IF;

		Retracting:
			IF RetractingTimer.Q THEN
				udp_data.state := state := Destabilizing;
			END_IF;

		Destabilizing:
			IF DestabilizingTimer.Q THEN
				udp_data.state := state := ReadyToRelease;
			END_IF;

		ReadyToRelease:
			IF fire_os THEN
				udp_data.state := state := Releasing;
				man_send := FALSE;
				man_open := FALSE;
			END_IF;

		Releasing:
			IF after OR NOT(fire) THEN
				udp_data.state := state := ReadyToWork;
			END_IF;

		RetryTransfer:
			IF RetryTimer.Q THEN
				udp_data.state := state := Stabilizing;
			END_IF;

	END_CASE;

	// Comm Logic
	udp_data.waiting := waiting := (
	udp_data.state = ReadyToRelease
	AND NOT(custom_send_lock)
	AND NOT(after)
	AND NOT(safety_zone)
	);

	udp_data.bring_ok := bring_ok := (
	udp_data.state = ReadyToWork
	AND NOT(arrive)
	AND NOT(going_to)
	AND NOT(custom_bring_lock)
	AND NOT(open)
	AND NOT(receive_signal)
	AND staticBagRailBringOk
	);

	IF udp_data.state = Releasing THEN
		loadcell.capture_weight_bool := TRUE;
	ELSE
		loadcell.capture_weight_bool := FALSE;
	END_IF;

		// Communication
	IF sling_ready THEN
		cat_binary := wash_com_cat;
		cust_binary := wash_com_cust;
		weight_binary := wash_com_wt;
	END_IF;
	IF NOT(sling_ready) THEN
		cat_binary := 0;
		cust_binary := 0;
		weight_binary := 0;
	END_IF;
	BIN_TO_BCD_INT_sc(RegisterIN:= cat_binary);
	cat_bcd := BIN_TO_BCD_INT_sc.RegisterOUT;
	BIN_TO_BCD_INT_cust(RegisterIN:= cust_binary);
	cust_bcd := BIN_TO_BCD_INT_cust.RegisterOUT;
	BIN_TO_BCD_INT_weight(RegisterIN:= weight_binary);
	weight_bcd := BIN_TO_BCD_INT_weight.RegisterOUT;

	// Insert
	IF going_to AND arrive THEN insert := TRUE; END_IF;

	// Output Control
	stb := (
	udp_data.state = Stabilizing
	OR udp_data.state = ReadyToTransfer
	OR udp_data.state = Transferring
	OR udp_data.state = LoadReceived
	OR udp_data.state = Extending
	OR udp_data.state = Clamping
	OR udp_data.state = Retracting
	);

	open := (
	udp_data.state = Transferring
	OR udp_data.state = LoadReceived
	OR udp_data.state = Extending
	);

	stp := udp_data.state = Releasing OR lift_stp;
	sling_ready := udp_data.state = ReadyToTransfer AND onoff AND NOT(halted) AND NOT(safety_zone);
	close := udp_data.state = Extending;

	// Speed reducing static always is 'unclampled'
	// Open and close also triggered in state machine
	static_open := TRUE;
	IF EDGEPOS(going_to) THEN static_close := FALSE; END_IF;

	// Control Timers
	ResetTimeout(IN := reset, PT := ResetTime);
	StabilizingTimer(IN := (udp_data.state = Stabilizing), PT := StabilizingTime);
	TransferringTimer(IN := (udp_data.state = Transferring), PT := TransferringTime);
	DestabilizingTimer(IN := (udp_data.state = Destabilizing), PT := DestabilizingTime);
	ExtendingTimer(IN := (udp_data.state = Extending), PT := ExtendingTime);
	RetractingTimer(IN := (udp_data.state = Retracting), PT := RetractingTime);
	ClampingTimer(IN := (udp_data.state = Clamping), PT := ClampingTime);
	RetryTimer(IN := (udp_data.state = RetryTransfer), PT := RetryTime);

	// Alarm Timers
	AlarmTimer(IN := fire, PT := (t#1s * rail_alarm_time));
	UnexpectedBagTimer(IN := (front AND rail_mt), PT := UnexpectedBagTime);
	MissingBagTimer(IN := (NOT(front) AND NOT(rail_mt)), PT := MissingBagTime);
	LoadNotDroppedTimer(IN:= (udp_data.state = Transferring), PT := AlmTime_LoadNotDropped);
	BagNotOpenTimer(IN:= ((udp_data.state = LoadReceived) AND empty_bag) , PT := BagNotOpenTime);

	udp_data.alarm := alarm := AlarmTimer.Q;
	udp_data.warning_com.0 := warning_com.0 := 0;//UnexpectedBagTimer.Q;
	udp_data.warning_com.1 := warning_com.1 := 0;//MissingBagTimer.Q;
	udp_data.warning_com.14 := warning_com.14 := sling_ready;

	// Rail Fault Handling.

	messages.Write := 0;
	//BAG_STUCK  -- NOT YET IMPLEMENTED
	IF UnexpectedBagTimer.Q   THEN messages.Write := BIT_SET(messages.Write,UNEXPECTED_BAG); END_IF;
	IF MissingBagTimer.Q      THEN messages.Write := BIT_SET(messages.Write,MISSING_BAG); END_IF;
	IF LoadNotDroppedTimer.Q  THEN messages.Write := BIT_SET(messages.Write,TOO_LONG_TO_TRANSFER); END_IF;
	IF BagNotOpenTimer.Q      THEN messages.Write := BIT_SET(messages.Write,BAG_NOT_OPEN); END_IF;
	IF ((udp_data.state = Stabilizing) AND StabilizingTimer.Q AND NOT empty_bag) THEN messages.Write := BIT_SET(messages.Write,BAG_EMPTY_PX); END_IF;

	// Always clear acknowledgements
	brsmemset(ADR(messages.Read[0]),0,SIZEOF(messages.Read));

END_FUNCTION_BLOCK
```

#### SupertrackDischarger.st
```iecst
(* TODO: Add your comment here *)
FUNCTION_BLOCK SupertrackDischarger

	messages ACCESS p_messages;
	loadcell ACCESS p_loadcell;

	// Debounce Inputs
	DBNC_front_timer(IN := front_raw, PT := DBNC_front_time);
	front := DBNC_front_timer.Q;

	DBNC_arrive_timer(IN := arrive_raw, PT := DBNC_arrive_time);
	arrive := DBNC_arrive_timer.Q;

	DBNC_after_timer(IN := after_raw, PT := DBNC_after_time);
	after := DBNC_after_timer.Q;

	// Device State Machine
	IF ResetTimeout.Q THEN
		udp_data.state := state := ReadyToWork;
		man_send := FALSE;
		man_open := FALSE;
	END_IF;
	IF udp_data.state = 0 THEN udp_data.state := state := ReadyToWork; END_IF;

	CASE udp_data.state OF
		ReadyToWork:
			IF NOT(rail_mt) AND front AND onoff AND NOT(halted) AND NOT(ResetTimeout.Q) THEN
				udp_data.state := state := Stabilizing;
			ELSIF man_send THEN
				udp_data.state := state := Destabilizing;
			END_IF;

		Stabilizing:
			static_close := FALSE;
			IF StabilizingTimer.Q THEN
				IF empty_bag OR (messages.Read[BAG_EMPTY_PX] = 1) THEN
					udp_data.state := state := ReadyToTransfer;
				ELSIF (messages.Read[BAG_EMPTY_PX] = 2) THEN
					udp_data.state := state := Destabilizing;
				END_IF;
			ELSIF NOT(onoff) THEN
				udp_data.state := state := ReadyToWork;
			ELSIF man_send THEN
				udp_data.state := state := Destabilizing;
			END_IF;

		ReadyToTransfer:
			IF open_signal OR open_pendant OR man_open THEN
				man_open := FALSE;
				udp_data.state := state := Transferring;
			ELSIF NOT(onoff) THEN
				udp_data.state := state := ReadyToWork;
			ELSIF man_send THEN
				udp_data.state := state := Destabilizing;
				man_send := FALSE;
			END_IF;

		Transferring:
			IF TransferringTimer.Q THEN
				static_close := TRUE;
			END_IF;
			IF receive_signal OR receive_pendant THEN
				udp_data.state := state := LoadReceived;
			ELSIF (messages.Read[TOO_LONG_TO_TRANSFER] > 0) THEN
				CASE messages.Read[TOO_LONG_TO_TRANSFER] OF
					1: //'retry_transfer'
						udp_data.state := state := RetryTransfer;
					2: //'send_bag_away'
						udp_data.state := state := Extending;
				END_CASE;
			ELSIF man_send THEN
				udp_data.state := state := Extending;
				man_send := FALSE;
			END_IF;

		LoadReceived:
			static_close := TRUE;
			IF empty_bag THEN // Bag hasn't opened
				CASE messages.Read[BAG_NOT_OPEN] OF
					1: //'retry_transfer'
						udp_data.state := state := RetryTransfer;
					2: //'send_bag_away'
						udp_data.state := state := Extending;
				END_CASE;
			ELSIF NOT(empty_bag) THEN
				udp_data.state := state := Extending;
			ELSIF man_send THEN
				udp_data.state := state := Extending;
				man_send := FALSE;
			END_IF;

		Extending:
			static_close := TRUE;
			IF ExtendingTimer.Q THEN
				udp_data.state := state := Clamping;
			END_IF;

		Clamping:
			IF ClampingTimer.Q THEN
				udp_data.state := state := Retracting;
			END_IF;

		Retracting:
			IF RetractingTimer.Q THEN
				udp_data.state := state := Destabilizing;
			END_IF;

		Destabilizing:
			IF DestabilizingTimer.Q THEN
				udp_data.state := state := ReadyToRelease;
			END_IF;

		ReadyToRelease:
			IF fire_os THEN
				udp_data.state := state := Releasing;
				man_send := FALSE;
				man_open := FALSE;
			END_IF;

		Releasing:
			IF after OR NOT(fire) THEN
				udp_data.state := state := ReadyToWork;
			END_IF;

		RetryTransfer:
			IF RetryTimer.Q THEN
				udp_data.state := state := Stabilizing;
			END_IF;

	END_CASE;

	// Comm Logic
	udp_data.waiting := waiting := (
	udp_data.state = ReadyToRelease
	AND NOT(custom_send_lock)
	AND NOT(after)
	AND NOT(safety_zone)
	);

	udp_data.bring_ok := bring_ok := (
	udp_data.state = ReadyToWork
	AND NOT(arrive)
	AND NOT(going_to)
	AND NOT(custom_bring_lock)
	AND NOT(open)
	AND NOT(receive_signal)
	);

	IF udp_data.state = Releasing THEN
		loadcell.capture_weight_bool := TRUE;
	ELSE
		loadcell.capture_weight_bool := FALSE;
	END_IF;

		// Communication
	IF sling_ready THEN
		cat_binary := wash_com_cat;
		cust_binary := wash_com_cust;
		weight_binary := wash_com_wt;
	END_IF;
	IF NOT(sling_ready) THEN
		cat_binary := 0;
		cust_binary := 0;
		weight_binary := 0;
	END_IF;
	BIN_TO_BCD_INT_sc(RegisterIN:= cat_binary);
	cat_bcd := BIN_TO_BCD_INT_sc.RegisterOUT;
	BIN_TO_BCD_INT_cust(RegisterIN:= cust_binary);
	cust_bcd := BIN_TO_BCD_INT_cust.RegisterOUT;
	BIN_TO_BCD_INT_weight(RegisterIN:= weight_binary);
	weight_bcd := BIN_TO_BCD_INT_weight.RegisterOUT;

	// Insert
	IF going_to AND arrive THEN insert := TRUE; END_IF;

	// Output Control
	stb := (
	udp_data.state = Stabilizing
	OR udp_data.state = ReadyToTransfer
	OR udp_data.state = Transferring
	OR udp_data.state = LoadReceived
	OR udp_data.state = Extending
	OR udp_data.state = Clamping
	OR udp_data.state = Retracting
	);

	open := (
	udp_data.state = Transferring
	OR udp_data.state = LoadReceived
	OR udp_data.state = Extending
	);

	stp := udp_data.state = Releasing OR lift_stp;
	sling_ready := udp_data.state = ReadyToTransfer AND onoff AND NOT(halted) AND NOT(safety_zone);
	close := udp_data.state = Extending;

	// Speed reducing static always is 'unclampled'
	// Open and close also triggered in state machine
	static_open := TRUE;
	IF EDGEPOS(going_to) THEN static_close := FALSE; END_IF;

	// Control Timers
	ResetTimeout(IN := reset, PT := ResetTime);
	StabilizingTimer(IN := (udp_data.state = Stabilizing), PT := StabilizingTime);
	TransferringTimer(IN := (udp_data.state = Transferring), PT := TransferringTime);
	DestabilizingTimer(IN := (udp_data.state = Destabilizing), PT := DestabilizingTime);
	ExtendingTimer(IN := (udp_data.state = Extending), PT := ExtendingTime);
	RetractingTimer(IN := (udp_data.state = Retracting), PT := RetractingTime);
	ClampingTimer(IN := (udp_data.state = Clamping), PT := ClampingTime);
	RetryTimer(IN := (udp_data.state = RetryTransfer), PT := RetryTime);

	// Alarm Timers
	AlarmTimer(IN := fire, PT := (t#1s * rail_alarm_time));
	UnexpectedBagTimer(IN := (front AND rail_mt), PT := UnexpectedBagTime);
	MissingBagTimer(IN := (NOT(front) AND NOT(rail_mt)), PT := MissingBagTime);
	LoadNotDroppedTimer(IN:= (udp_data.state = Transferring), PT := AlmTime_LoadNotDropped);
	BagNotOpenTimer(IN:= ((udp_data.state = LoadReceived) AND empty_bag) , PT := BagNotOpenTime);

	udp_data.alarm := alarm := AlarmTimer.Q;
	udp_data.warning_com.0 := warning_com.0 := 0;//UnexpectedBagTimer.Q;
	udp_data.warning_com.1 := warning_com.1 := 0;//MissingBagTimer.Q;
	udp_data.warning_com.14 := warning_com.14 := sling_ready;

	// Rail Fault Handling.

	messages.Write := 0;
	//BAG_STUCK  -- NOT YET IMPLEMENTED
	IF UnexpectedBagTimer.Q   THEN messages.Write := BIT_SET(messages.Write,UNEXPECTED_BAG); END_IF;
	IF MissingBagTimer.Q      THEN messages.Write := BIT_SET(messages.Write,MISSING_BAG); END_IF;
	IF LoadNotDroppedTimer.Q  THEN messages.Write := BIT_SET(messages.Write,TOO_LONG_TO_TRANSFER); END_IF;
	IF BagNotOpenTimer.Q      THEN messages.Write := BIT_SET(messages.Write,BAG_NOT_OPEN); END_IF;
	IF ((udp_data.state = Stabilizing) AND StabilizingTimer.Q AND NOT empty_bag) THEN messages.Write := BIT_SET(messages.Write,BAG_EMPTY_PX); END_IF;

	// Always clear acknowledgements
	brsmemset(ADR(messages.Read[0]),0,SIZEOF(messages.Read));

END_FUNCTION_BLOCK
```

#### SupertrackEasisort.st
```iecst
(* TODO: Add your comment here *)
FUNCTION_BLOCK SupertrackEasisort

	messages ACCESS p_messages;
	loadcell ACCESS p_loadcell;

	IF  udp_data.state = 0 THEN  udp_data.state := state := Resetting; END_IF;

	// Device State Machine
	IF reset THEN
		udp_data.state := state := Resetting;
		man_send := FALSE;
		purge := FALSE;
	END_IF;
	IF OverWeightTimer.Q AND (( udp_data.state = Loading) OR ( udp_data.state = NearWeight) OR ( udp_data.state = ReadyToRelease)) THEN
		 udp_data.state := state := OverWeight;
	END_IF;
	CASE  udp_data.state OF

		Resetting:
			IF ResettingTimer.Q THEN
			  udp_data.state := state := Loading;
			END_IF;

		Loading:
			IF purge THEN
              udp_data.state := state := OpenDoor;
            ELSIF NearWeightTimer.Q THEN
			  udp_data.state := state := NearWeight;
			ELSIF man_send THEN
			  udp_data.state := state := ReadyToRelease;
			END_IF;

		NearWeight:
			IF purge THEN
              udp_data.state := state := OpenDoor;
            ELSIF FullWeightTimer.Q THEN
			  udp_data.state := state := ReadyToRelease;
			ELSIF man_send THEN
			  udp_data.state := state := ReadyToRelease;
			END_IF;

		ReadyToRelease:
			IF fire_os THEN
				udp_data.state := state := OpenDoor;
			END_IF;

		OpenDoor:
			IF OpenDoorTimer.Q THEN
			  IF purge THEN
                udp_data.state := state := RunEmpty;
              ELSE
				udp_data.state := state := Releasing;
			  END_IF;
			END_IF;

		Releasing:
			IF after OR NOT(fire) THEN
			  udp_data.state := state := RunEmpty;
			END_IF;

		RunEmpty:
			IF EmptyWeightTimer.Q THEN
			  udp_data.state := state := CloseDoor;
			END_IF;

		CloseDoor:
			IF CloseDoorTimer.Q THEN
			  udp_data.state := state := Loading;
			  purge := FALSE;
			END_IF;

		OverWeight:
			IF (messages.Read[OVERWEIGHT] = 1) AND WeightOk.Q THEN
			  udp_data.state := state := Loading;
			END_IF;

	END_CASE;

	// Comm Logic
	udp_data.waiting := waiting := (
	(udp_data.state = ReadyToRelease)
	AND NOT custom_send_lock
	AND NOT after
	AND NOT safety_zone
	AND NOT loadcell.over_weight
	);

	// Inserts
	IF going_to AND arrive THEN insert := TRUE; END_IF;

	IF udp_data.state = NearWeight OR udp_data.state = Loading THEN
		loadcell.capture_weight_bool := TRUE;
	ELSE
		loadcell.capture_weight_bool := FALSE;
	END_IF;

	// Input Control
	man_send := FALSE; // Clear any manual send request if not on the right step
	IF man_send_button THEN
		man_send := TRUE;
	END_IF;

	// Output Control
	open := releasing :=  (
	udp_data.state = OpenDoor
	OR udp_data.state = Releasing
	OR udp_data.state = RunEmpty
	);

	run_conveyor  := (
	udp_data.state = Releasing
	OR udp_data.state = RunEmpty
	);

	red_light := (
	((loadcell.notify_weight AND SlowOnPulseTimer.Q)
	OR udp_data.state = ReadyToRelease
	OR udp_data.state = RunEmpty
	OR udp_data.state = CloseDoor
	OR udp_data.state = Releasing
	OR udp_data.state = Resetting
	AND NOT(loadcell.over_weight))
	OR (loadcell.over_weight AND FastOnPulseTimer.Q)
	);

	// Control Timers
	EmptyWeightTimer(IN:= loadcell.empty AND conveyor_running, PT:= EmptyWeightTime);
	NearWeightTimer(IN := (loadcell.near_weight), PT := NearWeightTime);
	FullWeightTimer(IN := (loadcell.full), PT := FullWeightTime);
	ResettingTimer(IN := (udp_data.state = Resetting), PT := ResettingTime);
	CloseDoorTimer(IN := (udp_data.state = CloseDoor), PT := CloseDoorTime);
	OpenDoorTimer(IN := udp_data.state = OpenDoor, PT:= OpenDoorTime);
	WeightOk(IN := (udp_data.state = OverWeight), PT:= WeightOkTime);

	FastOnPulseTimer(IN := NOT(FastOffPulseTimer.Q), PT := FastOnPulseTime);
	FastOffPulseTimer(IN := FastOnPulseTimer.Q, PT := FastOffPulseTime);
	SlowOnPulseTimer(IN := NOT(SlowOffPulseTimer.Q), PT := SlowOnPulseTime);
	SlowOffPulseTimer(IN := SlowOnPulseTimer.Q, PT := SlowOffPulseTime);

	// Alarm Timers
	AlarmTimer(IN := fire, PT := (t#1s * rail_alarm_time));
	OverWeightTimer(IN := (loadcell.over_weight AND NOT(rail_mt)), PT := OverWeightTime);

	udp_data.alarm := alarm := AlarmTimer.Q;

	messages.Write := 0;
	IF (udp_data.state = OverWeight)  THEN messages.Write := BIT_SET(messages.Write,OVERWEIGHT); END_IF;

	// Always clear acknowledgements
	brsmemset(ADR(messages.Read[0]),0,SIZEOF(messages.Read));

END_FUNCTION_BLOCK
```

#### SupertrackSlingToBelt.st
```iecst
(* TODO: Add your comment here *)
FUNCTION_BLOCK SupertrackSlingToBelt

	messages ACCESS p_messages;
	loadcell ACCESS p_loadcell;

	IF  udp_data.state = 0 THEN  udp_data.state := state := Resetting; END_IF;

	// Device State Machine
	IF reset THEN
		udp_data.state := state := Resetting;
		man_send := FALSE;
		purge := FALSE;
        cc_shut_top_os := FALSE;
        cc_open_top_os := FALSE;
	END_IF;

	IF OverWeightTimer.Q AND ((udp_data.state = Loading) OR (udp_data.state = NearWeight) OR (udp_data.state = FullWeight)) THEN
		udp_data.state := state := OverWeight;
	END_IF;

	CASE udp_data.state OF

		Resetting:
			IF ResettingTimer.Q THEN
				udp_data.state := state := TransitToLoading;
			END_IF;

		TransitToLoading:
			IF TransitToLoadingTimer.Q THEN
				udp_data.state := state := Loading;
			END_IF;

		Loading:
			IF NearWeightTimer.Q THEN
				udp_data.state := state := NearWeight;
			ELSIF man_send THEN
				udp_data.state := state := FullWeight;
			ELSIF purge AND NOT(safety_zone) THEN
              udp_data.state := state := Purge;
            ELSIF cc_shut_top_os THEN
                cc_shut_top_os := FALSE;
                udp_data.state := state := Buffering;
            END_IF;

		NearWeight:
			IF FullWeightTimer.Q THEN
				udp_data.state := state := FullWeight;
			ELSIF man_send THEN
				udp_data.state := state := FullWeight;
			ELSIF purge AND NOT(safety_zone) THEN
                  udp_data.state := state := Purge;
            ELSIF cc_shut_top_os THEN
                  cc_shut_top_os := FALSE;
                  udp_data.state := state := Buffering;
			END_IF;

		Buffering:
            cc_shut_top_os := FALSE;
            IF cc_open_top_os THEN
                cc_open_top_os := FALSE;
                udp_data.state := state := Resetting;
            ELSIF man_send THEN
                udp_data.state := state := FullWeight;
            ELSIF purge AND NOT(safety_zone) THEN
               udp_data.state := state := Purge;
            END_IF;

		FullWeight:
			IF CloseTopDoorTimer.Q THEN
				udp_data.state := state := ReadyToRelease;
				man_send := FALSE;
			END_IF;

		ReadyToRelease:
			IF fire_os THEN
				udp_data.state := state := Releasing;
			ELSIF OverWeightTimer.Q THEN
				udp_data.state := state := OverWeight;
			END_IF;

		Releasing:
			IF after OR NOT(fire) THEN
				udp_data.state := state := Resetting;
			END_IF;

		Purge:
			IF PurgeTimer.Q THEN
				udp_data.state := state := Resetting;
				purge := FALSE;
			END_IF;

		OverWeight:
			IF (messages.Read[OVERWEIGHT] = 1) AND WeightOk.Q THEN
				udp_data.state := state := Loading;
			END_IF;

	END_CASE;

	// Comm Logic
	udp_data.waiting := waiting := (
	udp_data.state = ReadyToRelease
	AND NOT(custom_send_lock)
	AND NOT(after)
	AND NOT(safety_zone)
	AND NOT (loadcell.over_weight)
	);

	// Inserts
	IF going_to AND arrive THEN insert := TRUE; END_IF;

	IF udp_data.state = NearWeight OR udp_data.state = Loading THEN
		loadcell.capture_weight_bool := TRUE;
	ELSE
		loadcell.capture_weight_bool := FALSE;
	END_IF;

	// Input Control
	IF man_send_button OR man_send_button_1 OR man_send_button_2 THEN
		man_send := TRUE;
	END_IF;

	// Output Control
	open_bottom := releasing := ReleaseDelayTimer.Q;
	close_top := (
	udp_data.state = FullWeight
	OR udp_data.state = ReadyToRelease
	OR udp_data.state = Releasing
	OR udp_data.state = Resetting
	OR udp_data.state = Purge
	OR udp_data.state = Buffering
	);

	green_light := (onoff) AND NOT(udp_data.state = FullWeight);

	red_light := (
	((loadcell.notify_weight AND SlowOnPulseTimer.Q)
	OR udp_data.state = FullWeight
	OR udp_data.state = ReadyToRelease
	OR udp_data.state = Releasing
	OR udp_data.state = Resetting
	AND NOT(loadcell.over_weight))
	OR (loadcell.over_weight AND FastOnPulseTimer.Q)
	);

	// Control Timers
	NearWeightTimer(IN := (loadcell.near_weight), PT := NearWeightTime);
	FullWeightTimer(IN := (loadcell.full), PT := FullWeightTime);
	CloseTopDoorTimer(IN := (udp_data.state = FullWeight), PT := CloseTopDoorTime);
	ResettingTimer(IN := (udp_data.state = Resetting), PT := ResettingTime);
	TransitToLoadingTimer(IN := (udp_data.state = TransitToLoading), PT := TransitToLoadingTime);
	ReleaseDelayTimer(IN := udp_data.state = Releasing, PT:= ReleaseDelayTime);
	PurgeTimer(IN := udp_data.state = Purge AND conveyor_rail_running AND NOT(safety_zone) AND open_bottom, PT:= PurgeTime);
	WeightOk(IN := (udp_data.state = OverWeight), PT:= WeightOkTime);

	FastOnPulseTimer(IN := NOT(FastOffPulseTimer.Q), PT := FastOnPulseTime);
	FastOffPulseTimer(IN := FastOnPulseTimer.Q, PT := FastOffPulseTime);
	SlowOnPulseTimer(IN := NOT(SlowOffPulseTimer.Q), PT := SlowOnPulseTime);
	SlowOffPulseTimer(IN := SlowOnPulseTimer.Q, PT := SlowOffPulseTime);

	// Alarm Timers
	AlarmTimer(IN := fire, PT := (t#1s * rail_alarm_time));
	udp_data.alarm := alarm := AlarmTimer.Q;
	OverWeightTimer(IN := (loadcell.over_weight AND NOT(rail_mt)), PT := OverWeightTime);

	messages.Write := 0;
	IF (state = OverWeight)  THEN messages.Write := BIT_SET(messages.Write,OVERWEIGHT); END_IF;

	// Always clear acknowledgements
	brsmemset(ADR(messages.Read[0]),0,SIZEOF(messages.Read));

END_FUNCTION_BLOCK
```

#### SupertrackSplitRailInxTracked.st
```iecst
(* TODO: Add your comment here *)
FUNCTION_BLOCK SupertrackSplitRailInxTracked

	messages ACCESS p_messages;

	  // Debounce Inputs
	DBNC_front_timer(IN := front_raw, PT := DBNC_front_time);
	front := DBNC_front_timer.Q;

	DBNC_arrive_timer(IN := arrive_raw, PT := DBNC_arrive_time);
	arrive := DBNC_arrive_timer.Q;

	DBNC_after_timer(IN := after_raw, PT := DBNC_after_time);
	after := DBNC_after_timer.Q;

	DBNC_before_timer(IN := before_raw, PT := DBNC_before_time);
	before := DBNC_before_timer.Q;

	// Device State Machine
	IF reset THEN udp_data.state := state := ReadyToRelease; END_IF;
	IF udp_data.state = 0 THEN udp_data.state := state := ReadyToRelease; END_IF;

	CASE udp_data.state OF
		ReadyToRelease:
			IF fire_os THEN
				udp_data.state := state := PrepareToRelease;
			END_IF;

		PrepareToRelease:
			IF TrolleyPrepareTimer.Q THEN
				udp_data.state := state := Releasing;
			END_IF;

		Releasing:
			IF after OR NOT(fire) THEN
				udp_data.state := state := ReadyToRelease;
			END_IF;

	END_CASE;

	// Comm Logic
	udp_data.waiting := waiting := (
	udp_data.state = ReadyToRelease
	AND front
	AND NOT(custom_send_lock)
	AND NOT(after)
	AND NOT(safety_zone)
	);

	udp_data.bring_ok := bring_ok := (
	NOT(before)
	AND NOT(arrive)
	AND NOT(going_to)
	AND NOT(custom_bring_lock)
	);

	IF going_to AND arrive THEN insert := TRUE; END_IF;

	// Input Control
	front_raw := front_a AND front_b;

	// Output Control
	inx := udp_data.state = PrepareToRelease;

	//Pressure Relief Outputs
	Pressure1Timer(IN := NOT(pressure_sensor_1) AND NOT(pressure_full_line_1), PT := Pressure1Time);
	Pressure2Timer(IN := NOT(pressure_sensor_2) AND NOT(pressure_full_line_2), PT := Pressure2Time);
	Pressure3Timer(IN := NOT(pressure_sensor_3) AND NOT(pressure_full_line_3), PT := Pressure3Time);
	Pressure4Timer(IN := NOT(pressure_sensor_4) AND NOT(pressure_full_line_4), PT := Pressure4Time);
	Pressure5Timer(IN := NOT(pressure_sensor_5) AND NOT(pressure_full_line_5), PT := Pressure5Time);

	pressure_stop_1 := Pressure1Timer.Q;
	pressure_stop_2 := Pressure2Timer.Q;
	pressure_stop_3 := Pressure3Timer.Q;
	pressure_stop_4 := Pressure4Timer.Q;
	pressure_stop_5 := Pressure5Timer.Q;

	// Output Switch Control
	IF SwInARTrig.Q THEN
		sw_in_a := TRUE;
	END_IF;

	IF before AND going_to THEN
		sw_in_a := FALSE;
		sw_in_b  := TRUE;
	END_IF;

	IF NOT(going_to) THEN
		sw_in_a := FALSE;
		sw_in_b  := FALSE;
	END_IF;

	IF SwOutARTrig.Q THEN
		sw_out_a := TRUE;
	END_IF;

	IF fire AND after THEN
		sw_out_a := FALSE;
		sw_out_b  := TRUE;
	END_IF;

	IF NOT(fire) THEN
		sw_out_a := FALSE;
		sw_out_b  := FALSE;
	END_IF;

	IF reset THEN
		sw_out_a := FALSE;
		sw_out_b  := FALSE;
	END_IF;

	// Control Triggers
	SwInARTrig(CLK := (going_to));
	SwOutARTrig(CLK := (fire));
	TrolleyPrepareTimer(IN := udp_data.state = PrepareToRelease, PT := TrolleyPrepareTime);

	// Alarm Timers
	AlarmTimer(IN := fire, PT := (t#1s * rail_alarm_time));
	UnexpectedBagTimer(IN := (arrive AND NOT(front) AND NOT(inx)), PT := UnexpectedBagTime);
	MissingBagTimer(IN := (NOT(front) AND NOT(rail_mt) AND NOT(inx)), PT := MissingBagTime);

	// Alarm Coms
	udp_data.alarm := alarm := AlarmTimer.Q;
	udp_data.warning_com.0 := warning_com.0 := UnexpectedBagTimer.Q;
	udp_data.warning_com.1 := warning_com.1 := MissingBagTimer.Q;

	messages.Write := 0;
	IF UnexpectedBagTimer.Q   THEN messages.Write := BIT_SET(messages.Write,UNEXPECTED_BAG); END_IF;
	IF MissingBagTimer.Q      THEN messages.Write := BIT_SET(messages.Write,MISSING_BAG); END_IF;

	// Always clear acknowledgements
	brsmemset(ADR(messages.Read[0]),0,SIZEOF(messages.Read));

END_FUNCTION_BLOCK
```

#### SupertrackSplitRailInxUnTracked.st
```iecst
(* TODO: Add your comment here *)
FUNCTION_BLOCK SupertrackSplitRailInxUnTracked

	messages ACCESS p_messages;

	// Debounce Inputs
	DBNC_front_timer(IN := front_raw, PT := DBNC_front_time);
	front := DBNC_front_timer.Q;

	DBNC_arrive_timer(IN := arrive_raw, PT := DBNC_arrive_time);
	arrive := DBNC_arrive_timer.Q;

	DBNC_after_timer(IN := after_raw, PT := DBNC_after_time);
	after := DBNC_after_timer.Q;

	DBNC_before_timer(IN := before_raw, PT := DBNC_before_time);
	before := DBNC_before_timer.Q;

	// Device State Machine
	IF reset THEN udp_data.state := state := ReadyToRelease; END_IF;
	IF udp_data.state = 0 THEN udp_data.state := state := ReadyToRelease; END_IF;

	CASE udp_data.state OF
		ReadyToRelease:
			IF fire_os THEN
				udp_data.state := state := PrepareToRelease;
			END_IF;

		PrepareToRelease:
			IF TrolleyPrepareTimer.Q THEN
				udp_data.state := state := Releasing;
			END_IF;

		Releasing:
			IF after OR NOT(fire) THEN
				udp_data.state := state := ReadyToRelease;
			END_IF;

	END_CASE;

	// Comm Logic
	udp_data.waiting := waiting := (
	udp_data.state = ReadyToRelease
	AND front
	AND NOT(custom_send_lock)
	AND NOT(after)
	AND NOT(safety_zone)
	);

	udp_data.bring_ok := bring_ok := (
	NOT(before)
	AND NOT(arrive)
	AND NOT(going_to)
	AND NOT(custom_bring_lock)
	);

	IF going_to AND arrive THEN insert := TRUE; END_IF;

	// Input Control
	front_raw := front_a AND front_b;

	// Output Control
	inx := udp_data.state = PrepareToRelease;

	//Pressure Relief Outputs
	Pressure1Timer(IN := NOT(pressure_sensor_1) AND NOT(pressure_full_line_1), PT := Pressure1Time);
	Pressure2Timer(IN := NOT(pressure_sensor_2) AND NOT(pressure_full_line_2), PT := Pressure2Time);
	Pressure3Timer(IN := NOT(pressure_sensor_3) AND NOT(pressure_full_line_3), PT := Pressure3Time);
	Pressure4Timer(IN := NOT(pressure_sensor_4) AND NOT(pressure_full_line_4), PT := Pressure4Time);
	Pressure5Timer(IN := NOT(pressure_sensor_5) AND NOT(pressure_full_line_5), PT := Pressure5Time);

	pressure_stop_1 := Pressure1Timer.Q;
	pressure_stop_2 := Pressure2Timer.Q;
	pressure_stop_3 := Pressure3Timer.Q;
	pressure_stop_4 := Pressure4Timer.Q;
	pressure_stop_5 := Pressure5Timer.Q;

	// Output Switch Control
	IF SwInARTrig.Q THEN
		sw_in_a := TRUE;
	END_IF;

	IF before AND going_to THEN
		sw_in_a := FALSE;
		sw_in_b  := TRUE;
	END_IF;

	IF NOT(going_to) THEN
		sw_in_a := FALSE;
		sw_in_b  := FALSE;
	END_IF;

	IF SwOutARTrig.Q THEN
		sw_out_a := TRUE;
	END_IF;

	IF fire AND after THEN
		sw_out_a := FALSE;
		sw_out_b  := TRUE;
	END_IF;

	IF NOT(fire) THEN
		sw_out_a := FALSE;
		sw_out_b  := FALSE;
	END_IF;

	IF reset THEN
		sw_out_a := FALSE;
		sw_out_b  := FALSE;
	END_IF;

	// Control Triggers
	SwInARTrig(CLK := (going_to));
	SwOutARTrig(CLK := (fire));
	TrolleyPrepareTimer(IN := udp_data.state = PrepareToRelease, PT := TrolleyPrepareTime);

	// Alarm Timers
	AlarmTimer(IN := fire, PT := (t#1s * rail_alarm_time));
	UnexpectedBagTimer(IN := (arrive AND NOT(front) AND NOT(inx)), PT := UnexpectedBagTime);

	// Alarm Coms
	udp_data.alarm := alarm := AlarmTimer.Q;
	udp_data.warning_com.0 := warning_com.0 := UnexpectedBagTimer.Q;

	messages.Write := 0;
	IF UnexpectedBagTimer.Q   THEN messages.Write := BIT_SET(messages.Write,UNEXPECTED_BAG); END_IF;

	// Always clear acknowledgements
	brsmemset(ADR(messages.Read[0]),0,SIZEOF(messages.Read));

END_FUNCTION_BLOCK
```

#### SupertrackStackerOffgoing.st
```iecst
(* TODO: Add your comment here *)
FUNCTION_BLOCK SupertrackStackerOffgoing

	messages ACCESS p_messages;

	  // Debounce Inputs
	DBNC_front_timer(IN := front_raw, PT := DBNC_front_time);
	front := DBNC_front_timer.Q;

	DBNC_arrive_timer(IN := arrive_raw, PT := DBNC_arrive_time);
	arrive := DBNC_arrive_timer.Q;

	DBNC_after_timer(IN := after_raw, PT := DBNC_after_time);
	after := DBNC_after_timer.Q;

	DBNC_before_timer(IN := before_raw, PT := DBNC_before_time);
	before := DBNC_before_timer.Q;

	DBNC_after_a_timer(IN := after_a_raw, PT := DBNC_after_a_time);
	after_a := DBNC_after_a_timer.Q;

	DBNC_after_b_timer(IN := after_b_raw, PT := DBNC_after_b_time);
	after_b := DBNC_after_b_timer.Q;

	// Device State Machine
	IF reset THEN udp_data.state := state := ReadyToWork; END_IF;
	IF udp_data.state = 0 THEN udp_data.state := state := ReadyToWork; END_IF;

	CASE udp_data.state OF
		ReadyToWork:
			IF NOT(rail_mt) AND front AND onoff AND NOT(halted) THEN
				udp_data.state := state := Extending;
			END_IF;

		Extending:
			IF ExtendingTimer.Q THEN
				udp_data.state := state := Retracting;
			END_IF;

		Retracting:
			IF RetractingTimer.Q THEN
				udp_data.state := state := ReadyToRelease;
			END_IF;

		ReadyToRelease:
			IF fire_os THEN
				udp_data.state := state := ReleasingFront;
			END_IF;

		ReleasingFront:
			IF after_a THEN
				udp_data.state := state := ReleasingRear;
			ELSIF NOT(fire) THEN
				udp_data.state := state := ReadyToWork;
			END_IF;

		ReleasingRear:
			IF after_b OR NOT(fire) THEN
				udp_data.state := state := Releasing;
			END_IF;

		Releasing:
			IF NOT(fire) OR after THEN
				udp_data.state := state := ReadyToWork;
			END_IF;

	END_CASE;

	// Comm Logic
	udp_data.waiting := waiting := (
	udp_data.state = ReadyToRelease
	AND front
	AND NOT(custom_send_lock)
	AND NOT(after_a)
	AND NOT(after_b)
	AND NOT(after)
	AND NOT(safety_zone)
	);

	udp_data.bring_ok := bring_ok := (
	udp_data.state = ReadyToWork
	AND NOT(arrive)
	AND NOT(going_to)
	AND NOT(front_a)
	AND NOT(front_b)
	AND NOT(level_arm)
	AND NOT(custom_bring_lock)
	);

	IF going_to AND arrive THEN insert := TRUE; END_IF;

	// Input Control
	arrive_raw := front_raw := front_a AND front_b;

	// Output Control
	level_arm := udp_data.state = Extending;
	stp_a := udp_data.state = ReleasingFront OR udp_data.state = ReleasingRear;
	stp_b := udp_data.state = ReleasingRear;
	switch := udp_data.state = ReleasingFront OR udp_data.state = ReleasingRear;
	reset_switch := udp_data.state = Releasing;

	// Control Timers
	ExtendingTimer(IN := (udp_data.state = Extending), PT := ExtendingTime);
	RetractingTimer(IN := (udp_data.state = Retracting), PT := RetractingTime);

	// Alarm Timers
	AlarmTimer(IN := fire, PT := (t#1s * rail_alarm_time));
	UnexpectedBagTimer(IN := ((arrive OR front) AND rail_mt AND NOT(stp_a OR stp_b)), PT := UnexpectedBagTime);
	MissingBagTimer(IN := (NOT(front) AND NOT(rail_mt) AND NOT(stp_a OR stp_b)), PT := MissingBagTime);

	// Alarm Coms
	udp_data.alarm := alarm := AlarmTimer.Q;
	udp_data.warning_com.0 := warning_com.0 := UnexpectedBagTimer.Q;
	udp_data.warning_com.1 := warning_com.1 := MissingBagTimer.Q;

	messages.Write := 0;
	IF UnexpectedBagTimer.Q   THEN messages.Write := BIT_SET(messages.Write,UNEXPECTED_BAG); END_IF;
	IF MissingBagTimer.Q      THEN messages.Write := BIT_SET(messages.Write,MISSING_BAG); END_IF;

	// Always clear acknowledgements
	brsmemset(ADR(messages.Read[0]),0,SIZEOF(messages.Read));

END_FUNCTION_BLOCK
```

#### SupertrackStackerOngoing.st
```iecst
(* TODO: Add your comment here *)
FUNCTION_BLOCK SupertrackStackerOngoing

	messages ACCESS p_messages;

	  // Debounce Inputs
	DBNC_front_timer(IN := front_raw, PT := DBNC_front_time);
	front := DBNC_front_timer.Q;

	DBNC_arrive_timer(IN := arrive_raw, PT := DBNC_arrive_time);
	arrive := DBNC_arrive_timer.Q;

	DBNC_after_timer(IN := after_raw, PT := DBNC_after_time);
	after := DBNC_after_timer.Q;

	DBNC_before_timer(IN := before_raw, PT := DBNC_before_time);
	before := DBNC_before_timer.Q;

	// Device State Machine
	IF reset THEN udp_data.state := state := ReadyToWork; END_IF;
	IF udp_data.state = 0 THEN udp_data.state := state := ReadyToWork; END_IF;

	CASE udp_data.state OF
		ReadyToWork:
			IF NOT(rail_mt) AND front AND onoff AND NOT(halted) THEN
				udp_data.state := state := Extending;
			END_IF;

		Extending:
			IF ExtendingTimer.Q THEN
				udp_data.state := state := Retracting;
			END_IF;

		Retracting:
			IF RetractingTimer.Q THEN
				udp_data.state := state := ReadyToRelease;
			END_IF;

		ReadyToRelease:
			IF fire_os THEN
				udp_data.state := state := Releasing;
			END_IF;

		Releasing:
			IF NOT(fire) OR after THEN
				udp_data.state := state := ReadyToWork;
			END_IF;
	END_CASE;

	// Comm Logic
	udp_data.waiting := waiting := (
	udp_data.state = ReadyToRelease
	AND front
	AND NOT(custom_send_lock)
	AND NOT(safety_zone)
	);

	udp_data.bring_ok := bring_ok := (
	udp_data.state = ReadyToWork
	AND NOT(arrive)
	AND NOT(going_to)
	AND NOT(tilt_arm)
	AND NOT(stp)
	AND NOT(ring_pusher)
	AND NOT(pusher)
	AND NOT(custom_bring_lock)
	AND NOT(safety_zone)
	);

	IF going_to AND arrive THEN insert := TRUE; END_IF;

	// Input Control
	arrive_raw := front_raw := front_a AND front_b;

	 // Output Control
	tilt_arm := udp_data.state = Extending;
	stp := udp_data.state = Releasing;
	pusher := PusherOnTimer.Q;
	ring_pusher :=  RingPusherTimer.Q;

	// Control Timers
	ExtendingTimer(IN := (udp_data.state = Extending), PT := ExtendingTime);
	RetractingTimer(IN := (udp_data.state = Retracting), PT := RetractingTime);
	PusherOnTimer(IN := udp_data.state = Releasing AND NOT(PusherOffTimer.Q), PT := PusherOnTime);
	PusherOffTimer(IN := udp_data.state = Releasing AND PusherOnTimer.Q, PT := PusherOffTime);

	RingPusherTimer(IN := udp_data.state = Extending, PT := RingPusherTime);

	// Output Switch Control
	IF SwInARTrig.Q THEN
		sw_in_a := TRUE;
	END_IF;

	IF before AND going_to THEN
		sw_in_a := FALSE;
		sw_in_b  := TRUE;
	END_IF;

	IF NOT(going_to) THEN
		sw_in_a := FALSE;
		sw_in_b  := FALSE;
	END_IF;

	IF SwOutARTrig.Q THEN
		sw_out_a := TRUE;
	END_IF;

	IF fire AND after THEN
		sw_out_a := FALSE;
		sw_out_b  := TRUE;
	END_IF;

	IF NOT(fire) THEN
		sw_out_a := FALSE;
		sw_out_b  := FALSE;
	END_IF;

	IF reset THEN
		sw_out_a := FALSE;
		sw_out_b  := FALSE;
	END_IF;

	// Control Triggers
	SwInARTrig(CLK := (going_to));
	SwOutARTrig(CLK := (fire));

	// Alarm Timers
	AlarmTimer(IN := fire, PT := (t#1s * rail_alarm_time));
	UnexpectedBagTimer(IN := ((arrive OR front) AND rail_mt AND NOT(stp)), PT := UnexpectedBagTime);
	MissingBagTimer(IN := (NOT(front) AND NOT(rail_mt) AND NOT(stp)), PT := MissingBagTime);

	// Alarm Coms
	udp_data.alarm := alarm := AlarmTimer.Q;
	udp_data.warning_com.0 := warning_com.0 := UnexpectedBagTimer.Q;
	udp_data.warning_com.1 := warning_com.1 := MissingBagTimer.Q;

	messages.Write := 0;
	IF UnexpectedBagTimer.Q   THEN messages.Write := BIT_SET(messages.Write,UNEXPECTED_BAG); END_IF;
	IF MissingBagTimer.Q      THEN messages.Write := BIT_SET(messages.Write,MISSING_BAG); END_IF;

	// Always clear acknowledgements
	brsmemset(ADR(messages.Read[0]),0,SIZEOF(messages.Read));

END_FUNCTION_BLOCK
```

#### SupertrackSplitRailStp.st
```iecst
(* TODO: Add your comment here *)
FUNCTION_BLOCK SupertrackSplitRailStp

	messages ACCESS p_messages;

	  // Debounce Inputs
	DBNC_front_timer(IN := front_raw, PT := DBNC_front_time);
	front := DBNC_front_timer.Q;

	DBNC_arrive_timer(IN := arrive_raw, PT := DBNC_arrive_time);
	arrive := DBNC_arrive_timer.Q;

	DBNC_after_timer(IN := after_raw, PT := DBNC_after_time);
	after := DBNC_after_timer.Q;

	DBNC_before_timer(IN := before_raw, PT := DBNC_before_time);
	before := DBNC_before_timer.Q;

	DBNC_after_a_timer(IN := after_a_raw, PT := DBNC_after_a_time);
	after_a := DBNC_after_a_timer.Q;

	DBNC_after_b_timer(IN := after_b_raw, PT := DBNC_after_b_time);
	after_b := DBNC_after_b_timer.Q;

	// Device State Machine
	IF reset THEN udp_data.state := state := ReadyToWork; END_IF;
	IF udp_data.state = 0 THEN udp_data.state := state := ReadyToWork; END_IF;

	CASE udp_data.state OF
		ReadyToWork:
			IF NOT(rail_mt) AND front AND onoff AND NOT(halted) THEN
				udp_data.state := state := ReadyToRelease;
			END_IF;

		ReadyToRelease:
			IF fire_os THEN
				udp_data.state := state := ReleasingFront;
			END_IF;

		ReleasingFront:
			IF after_a THEN
				udp_data.state := state := ReleasingRear;
			ELSIF NOT(fire) THEN
				udp_data.state := state := ReadyToWork;
			END_IF;

		ReleasingRear:
			IF after_b OR NOT(fire) THEN
				udp_data.state := state := ReadyToWork;
			END_IF;
	END_CASE;

	// Comm Logic
	udp_data.waiting := waiting := (
	udp_data.state = ReadyToRelease
	AND front
	AND NOT(custom_send_lock)
	AND NOT(after_b)
	AND NOT(after)
	AND NOT(safety_zone)
	);

	udp_data.bring_ok := bring_ok := (
	udp_data.state = ReadyToWork
	AND NOT(before)
	AND NOT(arrive)
	AND NOT(front_a)
	AND NOT(front_b)
	AND NOT(going_to)
	AND NOT(custom_bring_lock)
	);

	IF going_to AND arrive THEN insert := TRUE; END_IF;

	// Input Control
	arrive_raw := front_raw := front_a AND front_b;

	// Output Control
	stp := udp_data.state = ReleasingFront OR udp_data.state = ReleasingRear;
	stp_a := udp_data.state = ReleasingFront OR udp_data.state = ReleasingRear;
	stp_b := udp_data.state = ReleasingRear;

	// Output Switch Control
	IF SwInARTrig.Q THEN
		sw_in_a := TRUE;
	END_IF;

	IF before AND going_to THEN
		sw_in_a := FALSE;
		sw_in_b  := TRUE;
	END_IF;

	IF NOT(going_to) THEN
		sw_in_a := FALSE;
		sw_in_b  := FALSE;
	END_IF;

	IF SwOutARTrig.Q THEN
		sw_out_a := TRUE;
	END_IF;

	IF fire AND after THEN
		sw_out_a := FALSE;
		sw_out_b  := TRUE;
	END_IF;

	IF NOT(fire) THEN
		sw_out_a := FALSE;
		sw_out_b  := FALSE;
	END_IF;

	IF reset THEN
		sw_out_a := FALSE;
		sw_out_b  := FALSE;
	END_IF;

	// Control Triggers
	SwInARTrig(CLK := (going_to));
	SwOutARTrig(CLK := (fire));

	// Alarm Timers
	AlarmTimer(IN := fire, PT := (t#1s * rail_alarm_time));
	UnexpectedBagTimer(IN := (arrive AND NOT(front) AND NOT(stp OR stp_a OR stp_b)), PT := UnexpectedBagTime);
	MissingBagTimer(IN := (NOT(front) AND NOT(rail_mt) AND NOT(stp OR stp_a OR stp_b)), PT := MissingBagTime);

	// Alarm Coms
	udp_data.alarm := alarm := AlarmTimer.Q;
	udp_data.warning_com.0 := warning_com.0 := UnexpectedBagTimer.Q;
	udp_data.warning_com.1 := warning_com.1 := MissingBagTimer.Q;

	messages.Write := 0;
	IF UnexpectedBagTimer.Q   THEN messages.Write := BIT_SET(messages.Write,UNEXPECTED_BAG); END_IF;
	IF MissingBagTimer.Q      THEN messages.Write := BIT_SET(messages.Write,MISSING_BAG); END_IF;

	// Always clear acknowledgements
	brsmemset(ADR(messages.Read[0]),0,SIZEOF(messages.Read));

END_FUNCTION_BLOCK
```

#### SupertrackRotaryTrf.st
```iecst
(* TODO: Add your comment here *)
FUNCTION_BLOCK SupertrackRotaryTrf

	messages ACCESS p_messages;

	// Debounce Inputs
	DBNC_after_timer(IN := after_raw, PT := DBNC_after_time);
	after := DBNC_after_timer.Q;

	DBNC_before_timer(IN := before_raw, PT := DBNC_before_time);
	before := DBNC_before_timer.Q;

	// Device State Machine
	IF reset THEN udp_data.state := state := Reset; END_IF;
	IF udp_data.state = 0 THEN udp_data.state := state := Reset; END_IF;

	CASE udp_data.state OF

		Reset: // Check the points are straight
			IF onoff AND NOT(halted) THEN
				IF ton_rotated.Q AND NOT rail_mt THEN
					udp_data.state := state := SettleOnPoints;
				ELSIF rail_mt AND NOT front_a AND NOT front_b THEN
					udp_data.state := state := ReadyToReceive;
				ELSIF front_a AND NOT rail_mt THEN
					udp_data.state := state := ReadyToRelease;
				END_IF;
			END_IF;

		ReadyToReceive: // stp b is open
			IF going_to THEN
				udp_data.state := state := ReceivingStraight;
			ELSIF ton_request_rotate.Q THEN // Requested to go to rotate position
				udp_data.state := state := MoveToRotate;
			END_IF;

		ReceivingStraight: //Bag is on its way
			IF arrive THEN
				udp_data.state := state := ReadyToRelease;
			END_IF;

		MoveToRotate: // Move to "in" position
			IF ton_rotated.Q THEN
				udp_data.state := state := SettleOnPoints;
			END_IF;

		SettleOnPoints:  //Wait for bag to arrive a and b closed
			IF ton_settledOnPoints.Q THEN
				udp_data.state := state := MoveToStraight;
			END_IF;

		MoveToStraight:
			IF ton_straight.Q THEN
				udp_data.state := state := ReadyToRelease;
			END_IF;

		ReadyToRelease:
			IF fire_os THEN
				udp_data.state := state := Releasing;
			END_IF;

		Releasing:
			IF after OR NOT(fire) THEN
				udp_data.state := state := Reset;
			END_IF;

	END_CASE;

	// Comm Logic
	udp_data.waiting := waiting := (
	udp_data.state = ReadyToRelease
	AND ton_straight.Q
	AND NOT(custom_send_lock)
	AND NOT(after)
	AND NOT(safety_zone)
	);

	udp_data.bring_ok := bring_ok := (
	((udp_data.state = ReadyToReceive) AND ton_straight.Q AND NOT request_rotate) OR
	((udp_data.state = SettleOnPoints) AND ton_rotated.Q)
	AND NOT(front_a)
	AND NOT(front_b)
	AND NOT(going_to)
	AND NOT(custom_bring_lock)
	);

	ton_request_rotate(IN:= request_rotate, PT:= requestRotateTime);

	IF going_to AND arrive THEN insert := TRUE; END_IF;

	// Input Control
	arrive := arrive_raw OR front_a;
	front := front_a OR front_b;

	// Output Control
	stp_a := (udp_data.state = Releasing) AND ton_straight.Q;
	stp_b := ((udp_data.state = Releasing) OR (udp_data.state = ReceivingStraight)) AND ton_straight.Q;

	switch := (
	(udp_data.state = MoveToRotate)
	OR (udp_data.state = SettleOnPoints)
	);// AND NOT ton_rotated.Q;

	reset_switch  := (
	(udp_data.state = ReadyToReceive)
	OR (udp_data.state = ReceivingStraight)
	OR (udp_data.state = MoveToStraight)
	OR (udp_data.state = ReadyToRelease)
	OR (udp_data.state = Releasing)
	);// AND NOT ton_straight.Q;

	ton_rotated(IN:= sw_in_a AND sw_in_b, PT:= rotateTime);
	ton_straight(IN:= sw_out_a AND sw_out_b, PT:= rotateTime);
	ton_settledOnPoints(IN:= front_a AND front_b, PT:= settleTime);

	// Alarm Timers
	AlarmTimer(IN := fire, PT := (t#1s * rail_alarm_time));
	UnexpectedBagTimer(IN := (arrive AND NOT(front)), PT := UnexpectedBagTime);
	MissingBagTimer(IN := (NOT(front) AND NOT(rail_mt)), PT := MissingBagTime);

	// Alarm Coms
	udp_data.alarm := alarm := AlarmTimer.Q;
	udp_data.warning_com.0 := warning_com.0 := UnexpectedBagTimer.Q;
	udp_data.warning_com.1 := warning_com.1 := MissingBagTimer.Q;

	messages.Write := 0;
	IF UnexpectedBagTimer.Q   THEN messages.Write := BIT_SET(messages.Write,UNEXPECTED_BAG); END_IF;
	IF MissingBagTimer.Q      THEN messages.Write := BIT_SET(messages.Write,MISSING_BAG); END_IF;

	// Always clear acknowledgements
	brsmemset(ADR(messages.Read[0]),0,SIZEOF(messages.Read));

END_FUNCTION_BLOCK
```

#### SupertrackRotaryTrn.st
```iecst
(* TODO: Add your comment here *)
FUNCTION_BLOCK SupertrackRotaryTrn

	messages ACCESS p_messages;

	  // Debounce Inputs
	DBNC_after_timer(IN := after_raw, PT := DBNC_after_time);
	after := DBNC_after_timer.Q;

	DBNC_before_timer(IN := before_raw, PT := DBNC_before_time);
	before := DBNC_before_timer.Q;

	// Device State Machine
	IF reset THEN udp_data.state := state := Reset; END_IF;
	IF udp_data.state = 0 THEN udp_data.state := state := Reset; END_IF;

	CASE udp_data.state OF

		Reset: //Always move to straight then decide what to do
			IF onoff AND NOT(halted) THEN
				IF ton_straight.Q AND NOT rail_mt THEN
					udp_data.state := state := SettleOnPoints;
				ELSIF ton_straight.Q AND rail_mt AND NOT front_a AND NOT front_b THEN
					udp_data.state := state := ReadyToReceive;
				END_IF;
			END_IF;

		ReadyToReceive: // stp b is open wait for bag to arrive.
			IF going_to THEN
				udp_data.state := state := Receiving;
			END_IF;

		Receiving: //Bag is on its way  stp b is open wait for bag to arrive.
			IF arrive THEN
				udp_data.state := state := SettleOnPoints;
			END_IF;

		SettleOnPoints:  //Wait for bag to arrive a and b closed
			IF ton_settledOnPoints.Q THEN
				udp_data.state := state := ReadyToRelease;
			END_IF;

		ReadyToRelease:// Decide where to send bag - Waiting for straight rail is on.
			IF fire_os THEN
				udp_data.state := state := ReleasingStraight;
			ELSIF request_rotate THEN
				udp_data.state := state := MoveToRotate;
			END_IF;

		MoveToRotate: // Move to "in" position
			IF ton_rotated.Q THEN
				udp_data.state := state := ReadyToReleaseRotate;
			END_IF;

		ReadyToReleaseRotate:
			IF fire_os THEN
				udp_data.state := state := ReleasingRotate;
			END_IF;

		ReleasingStraight:
			IF after OR NOT(fire) THEN
				udp_data.state := state := Reset;
			END_IF;

		ReleasingRotate:
			IF after OR NOT(fire) THEN
				udp_data.state := state := Reset;
			END_IF;

	END_CASE;

	// Comm Logic
	udp_data.waiting := waiting := (
	(((udp_data.state = ReadyToRelease) AND ton_straight.Q)
	OR ((udp_data.state = ReadyToReleaseRotate) AND ton_rotated.Q))
	AND NOT(custom_send_lock)
	AND NOT(after)
	AND NOT(safety_zone)
	);

	udp_data.bring_ok := bring_ok := (
	(udp_data.state = ReadyToReceive)
	AND ton_straight.Q
	AND NOT(front_a)
	AND NOT(front_b)
	AND NOT(going_to)
	AND NOT(custom_bring_lock)
	);

	IF going_to AND arrive THEN insert := TRUE; END_IF;

	// Input Control
	arrive := arrive_raw;
	front := front_a OR front_b;

	// Output Control
	stp_a := (
	((udp_data.state = ReleasingStraight) AND ton_straight.Q)
	OR ((udp_data.state = ReleasingRotate) AND ton_rotated.Q)
	);

	stp_b := (
	((udp_data.state = ReleasingStraight) AND ton_straight.Q)
	OR ((udp_data.state = ReleasingRotate) AND ton_rotated.Q)
	OR (udp_data.state = ReadyToReceive)
	OR (udp_data.state = Receiving)
	);

	rotate := (
	(udp_data.state = MoveToRotate)
	OR (udp_data.state = ReadyToReleaseRotate)
	OR (udp_data.state = ReleasingRotate)
	);

	switch := rotate;
	reset_switch  := NOT rotate;

	ton_straight(IN:= sw_in_a AND sw_in_b, PT:= rotateTime);
	ton_rotated(IN:= sw_out_a AND sw_out_b, PT:= rotateTime);
	ton_settledOnPoints(IN:= front_a AND front_b, PT:= settleTime);

	// Alarm Timers
	AlarmTimer(IN := fire, PT := (t#1s * rail_alarm_time));
	UnexpectedBagTimer(IN := (arrive AND NOT(front)), PT := UnexpectedBagTime);
	MissingBagTimer(IN := (NOT(front) AND NOT(rail_mt)), PT := MissingBagTime);

	// Alarm Coms
	udp_data.alarm := alarm := AlarmTimer.Q;
	udp_data.warning_com.0 := warning_com.0 := UnexpectedBagTimer.Q;
	udp_data.warning_com.1 := warning_com.1 := MissingBagTimer.Q;

	messages.Write := 0;
	IF UnexpectedBagTimer.Q   THEN messages.Write := BIT_SET(messages.Write,UNEXPECTED_BAG); END_IF;
	IF MissingBagTimer.Q      THEN messages.Write := BIT_SET(messages.Write,MISSING_BAG); END_IF;

	// Always clear acknowledgements
	brsmemset(ADR(messages.Read[0]),0,SIZEOF(messages.Read));

END_FUNCTION_BLOCK
```

#### SupertrackIncline.st
```iecst
(* TODO: Add your comment here *)
FUNCTION_BLOCK SupertrackIncline

	messages ACCESS p_messages;

	  // Debounce Inputs
	DBNC_arrive_timer(IN := arrive_raw, PT := DBNC_arrive_time);
	arrive := DBNC_arrive_timer.Q;

	DBNC_after_timer(IN := after_raw, PT := DBNC_after_time);
	after := DBNC_after_timer.Q;

	// Device State Machine
	IF reset AND rail_mt THEN
		udp_data.state := state := AlignLift;
	ELSIF reset AND NOT(rail_mt) THEN
		udp_data.state := state := ReadyToWork;
	END_IF;
	IF udp_data.state = 0 THEN udp_data.state := state := AlignLift; END_IF;

	CASE udp_data.state OF
		ReadyToWork:
			IF NOT(rail_mt) AND onoff AND NOT(halted) THEN
				udp_data.state := state := ReadyToRelease;
			END_IF;

		ReadyToRelease:
			IF fire_os THEN
				udp_data.state := state := Releasing;
			END_IF;

		Releasing:
			IF after OR NOT(fire) THEN
				udp_data.state := state := AlignLift;
			END_IF;

		AlignLift:
			IF paddle_sensor THEN
				udp_data.state := state := ReadyToWork;
			END_IF;
	END_CASE;

	// Comm Logic
	udp_data.waiting := waiting := (
	udp_data.state = ReadyToRelease
	AND rail_full
	AND NOT(custom_send_lock)
	AND NOT(after)
	AND NOT(safety_zone)
	);

	udp_data.bring_ok := bring_ok := (
	udp_data.state = ReadyToWork
	AND rail_mt
	AND NOT(arrive)
	AND NOT(going_to)
	AND NOT(custom_bring_lock)
	);

	IF going_to AND arrive THEN insert := TRUE; END_IF;

	// Output Control
	run_slant := ((udp_data.state = Releasing OR udp_data.state = AlignLift) AND onoff);

	// Alarm Timers
	AlarmTimer(IN := fire, PT := (t#1s * rail_alarm_time));
	UnexpectedBagTimer(IN := (arrive AND rail_mt AND NOT(run_slant)), PT := UnexpectedBagTime);

	// Alarm Coms
	udp_data.alarm := alarm := AlarmTimer.Q;
	udp_data.warning_com.0 := warning_com.0 := UnexpectedBagTimer.Q;

	messages.Write := 0;
	IF UnexpectedBagTimer.Q   THEN messages.Write := BIT_SET(messages.Write,UNEXPECTED_BAG); END_IF;

	// Always clear acknowledgements
	brsmemset(ADR(messages.Read[0]),0,SIZEOF(messages.Read));

END_FUNCTION_BLOCK
```

#### SupertrackStp.st
```iecst
(* TODO: Add your comment here *)
FUNCTION_BLOCK SupertrackStp

	messages ACCESS p_messages;
	loadcell ACCESS p_loadcell;

	  // Debounce Inputs
	DBNC_front_timer(IN := front_raw, PT := DBNC_front_time);
	front := DBNC_front_timer.Q;

	DBNC_arrive_timer(IN := arrive_raw, PT := DBNC_arrive_time);
	arrive := DBNC_arrive_timer.Q;

	DBNC_after_timer(IN := after_raw, PT := DBNC_after_time);
	after := DBNC_after_timer.Q;

	// Device State Machine
	IF reset THEN udp_data.state := state := ReadyToWork; END_IF;
	IF udp_data.state = 0 THEN udp_data.state := state := ReadyToWork; END_IF;

	CASE udp_data.state OF
		ReadyToWork:
			IF NOT(rail_mt) AND front AND onoff AND NOT(halted) THEN
				udp_data.state := state := ReadyToRelease;
			END_IF;

		ReadyToRelease:
			IF fire_os THEN
				udp_data.state := state := Releasing;
			ELSIF EmptyTimeoutTimer.Q THEN
				udp_data.state := state := ReadyToWork;
			END_IF;

		Releasing:
			IF after OR NOT(fire) THEN
				udp_data.state := state := ReadyToWork;
			END_IF;
	END_CASE;

	// Comm Logic
	udp_data.waiting := waiting := (
	udp_data.state = ReadyToRelease
	AND front
	AND NOT(custom_send_lock)
	AND NOT(after)
	AND NOT(safety_zone)
	);

	udp_data.bring_ok := bring_ok := (
	udp_data.state = ReadyToWork
	AND NOT(arrive)
	AND NOT(going_to)
	AND NOT(custom_bring_lock)
	);

	IF going_to AND arrive THEN insert := TRUE; END_IF;

	// Weight Comm
	IF udp_data.state = ReadyToWork OR udp_data.state = ReadyToRelease THEN
		loadcell.capture_weight_bool := TRUE;
	ELSE
		loadcell.capture_weight_bool := FALSE;
	END_IF;

	// Output Control
	stp := udp_data.state = Releasing;

	// Control Timers
	EmptyTimeoutTimer(IN := udp_data.state = ReadyToRelease AND rail_mt AND NOT(front) AND NOT(arrive), PT := EmptyTimeoutTime);

	// Alarm Timers
	AlarmTimer(IN := fire, PT := (t#1s * rail_alarm_time));
	UnexpectedBagTimer(IN := (front AND rail_mt AND NOT(stp)), PT := UnexpectedBagTime);
	MissingBagTimer(IN := (NOT(front) AND NOT(rail_mt) AND NOT(stp)), PT := MissingBagTime);

	// Alarm Coms
	udp_data.alarm := alarm := AlarmTimer.Q;
	udp_data.warning_com.0 := warning_com.0 := UnexpectedBagTimer.Q;
	udp_data.warning_com.1 := warning_com.1 := MissingBagTimer.Q;

	messages.Write := 0;
	IF UnexpectedBagTimer.Q   THEN messages.Write := BIT_SET(messages.Write,UNEXPECTED_BAG); END_IF;
	IF MissingBagTimer.Q      THEN messages.Write := BIT_SET(messages.Write,MISSING_BAG); END_IF;

	// Always clear acknowledgements
	brsmemset(ADR(messages.Read[0]),0,SIZEOF(messages.Read));

END_FUNCTION_BLOCK
```

#### SupertrackStaticBag.st
```iecst
(* TODO: Add your comment here *)
FUNCTION_BLOCK SupertrackStaticBag

	messages ACCESS p_messages;

	// Device State Machine
	IF reset THEN
		IF rail_mt THEN
			udp_data.state := state := ReadyToReceive;
		ELSE
			udp_data.state := state := Loaded;
		END_IF;
	END_IF;
	IF udp_data.state = 0 THEN udp_data.state := state := ReadyToReceive; END_IF;

	CASE udp_data.state OF
		Closed:
			IF input_enabled AND NOT(safety_zone) AND NOT(halted) THEN
				udp_data.state := state := ReadyToReceive;
			END_IF;

		ReadyToReceive:
			IF man_send THEN
				udp_data.state := state := Receiving;
			ELSIF NOT(input_enabled) OR safety_zone OR halted THEN
				udp_data.state := state := Closed;
			ELSIF NOT(rail_mt) THEN
				udp_data.state := state := Loaded;
			END_IF;

		Receiving:
			IF ReceivingTimer.Q THEN udp_data.state := state := Clamping; END_IF;

		Clamping:
			IF ClampingTimer.Q THEN udp_data.state := state := Loaded; END_IF;

		Loaded:
			IF NOT(halted) AND NOT(safety_zone) AND NOT(stopped) THEN
				udp_data.state := state := ReadyToTransfer;
			END_IF;

		ReadyToTransfer:
			IF open_signal OR man_open OR open_pendant THEN
				delete_latch := TRUE;
				udp_data.state := state := Unclamping;
			ELSIF halted OR stopped OR safety_zone THEN
				udp_data.state := state := Loaded;
			ELSIF rail_mt THEN
				udp_data.state := state := Closed;
			END_IF;

		Unclamping:
			IF UnclampingTimer.Q THEN udp_data.state := state := Transferring; END_IF;

		Transferring:
			IF man_send THEN udp_data.state := state := Closing; END_IF;

		Closing:
			IF ClosingTimer.Q AND NOT(delete_latch) THEN udp_data.state := state := ReadyToReceive; END_IF;

	END_CASE;

	// Output Control
	clamp := (
	udp_data.state = Unclamping
	OR udp_data.state = Transferring
	OR udp_data.state = Closing
	OR udp_data.state = Closed
	OR udp_data.state = ReadyToReceive
	OR udp_data.state = Receiving
	);

	open := udp_data.state = Transferring;

	// Control Timers
	ReceivingTimer(IN := (udp_data.state = Receiving), PT := ReceivingTime);
	ClampingTimer(IN := (udp_data.state = Clamping), PT := ClampingTime);
	UnclampingTimer(IN := (udp_data.state = Unclamping), PT := UnclampingTime);
	ClosingTimer(IN := (udp_data.state = Closing), PT := ClosingTime);

	// Comm Logic
	bring_ok := udp_data.state = Closing OR udp_data.state = Closed OR udp_data.state = ReadyToReceive;
	waiting := FALSE;
	man_open := man_send := FALSE;
	sling_ready := udp_data.state = ReadyToTransfer;
	dischargerRailReceiveSignal := udp_data.state = Clamping;

	IF rail_mt THEN delete_latch := FALSE; END_IF;

	udp_data.alarm := alarm := FALSE;
	udp_data.warning_com.0 := warning_com.0 := FALSE;
	udp_data.warning_com.1 := warning_com.1 := FALSE;
	udp_data.warning_com.12 := warning_com.12 := delete_latch;
	udp_data.warning_com.14 := warning_com.14 := sling_ready;

	//messages.Write := 0;
	//IF UnexpectedBagTimer.Q   THEN messages.Write := BIT_SET(messages.Write,UNEXPECTED_BAG); END_IF;
	//IF MissingBagTimer.Q      THEN messages.Write := BIT_SET(messages.Write,MISSING_BAG); END_IF;

	// Always clear acknowledgements
	//brsmemset(ADR(messages.Read[0]),0,SIZEOF(messages.Read));

END_FUNCTION_BLOCK
```

#### SupertrackBeltTransfer.st
```iecst
(* TODO: Add your comment here *)
FUNCTION_BLOCK SupertrackBeltTransfer

	messages ACCESS p_messages;

	  // Debounce Inputs
	DBNC_front_timer(IN := front_raw, PT := DBNC_front_time);
	front := DBNC_front_timer.Q;

	DBNC_arrive_timer(IN := arrive_raw, PT := DBNC_arrive_time);
	arrive := DBNC_arrive_timer.Q;

	DBNC_after_timer(IN := after_raw, PT := DBNC_after_time);
	after := DBNC_after_timer.Q;

	// Device State Machine
	IF reset THEN
		udp_data.state := state := ReadyToWork;
		halted := halt := FALSE;
	END_IF;

	IF udp_data.state = 0 THEN udp_data.state := state := ReadyToWork; END_IF;

	CASE udp_data.state OF
		ReadyToWork:
			IF NOT(rail_mt) AND NOT(halted) THEN
				udp_data.state := state := RunToFront;
			END_IF;

		RunToFront:
			IF NOT(front) THEN
				udp_data.state := state := ReadyToRelease;
			END_IF;

		ReadyToRelease:
			IF fire_os THEN
				udp_data.state := state := Releasing;
			END_IF;

		Releasing:
			IF after OR NOT(fire) THEN
				udp_data.state := state := ClearBelt;
			END_IF;

		ClearBelt:
			IF ClearBeltTimer.Q THEN
				udp_data.state := state := ReadyToWork;
			END_IF;
	END_CASE;

	// Comm Logic
	udp_data.waiting := waiting := (
	udp_data.state = ReadyToRelease
	AND NOT(custom_send_lock)
	AND NOT(after)
	AND NOT(safety_zone)
	);

	udp_data.bring_ok := bring_ok := (
	udp_data.state = ReadyToWork
	AND arrive
	AND front
	AND NOT(custom_bring_lock)
	AND NOT(going_to)
	AND NOT(ClearWarningTimer.Q)
	);

	IF going_to AND NOT(arrive) THEN insert := TRUE; END_IF;

	releasing := (
	udp_data.state = Releasing
	OR udp_data.state = ClearBelt
	);

	// Output Control
	run_conveyor := (
	NOT(halted) AND NOT halt
	AND (
	udp_data.state = Releasing
	OR udp_data.state = ClearBelt
	OR udp_data.state = RunToFront
	OR (going_to AND front AND (udp_data.state = ReadyToWork))
	));

	clear_belt := udp_data.state = Releasing OR udp_data.state = ClearBelt;

	//Control Timers
	MaximumBeltRunningTime(IN:=(run_conveyor AND conveyor_running), PT := MaximumRunningTime);
	ClearWarningTimer(IN:= warning_com.13, PT := ClearWarningTime);
	ClearBeltTimer(IN := (udp_data.state = ClearBelt AND arrive AND NOT receiving AND conveyor_running AND front AND NOT(fire)), PT := ClearBeltTime);
	IF MaximumBeltRunningTime.Q THEN
		halt := TRUE;
	END_IF;

	// Alarm Timers
	AlarmTimer(IN := fire, PT := (t#1s * rail_alarm_time));
	UnexpectedBagTimer(IN := (NOT front AND ((rail_mt AND (udp_data.state <> ClearBelt)) OR (conveyor_running AND (udp_data.state = ClearBelt)))) , PT := UnexpectedBagTime);
	MissingBagTimer(IN := (front AND NOT(rail_mt)), PT := MissingBagTime);

	// Alarm Coms
	udp_data.alarm := alarm := AlarmTimer.Q;
	udp_data.warning_com.0 := warning_com.0 := 0;//UnexpectedBagTimer.Q;
	udp_data.warning_com.1 := warning_com.1 := 0;//MissingBagTimer.Q;

	//Rail Messages
	messages.Write := 0;
	//BAG_STUCK # not yet implemented
	IF UnexpectedBagTimer.Q THEN messages.Write := BIT_SET(messages.Write,UNEXPECTED_BAG); END_IF;
	IF MissingBagTimer.Q THEN messages.Write := BIT_SET(messages.Write,MISSING_BAG); END_IF;
	IF halt THEN  messages.Write := BIT_SET(messages.Write,EXCEED_RUN_TIME); END_IF;

	CASE messages.Read[EXCEED_RUN_TIME] OF
		1: //They want to continue running
			halt := 0;
		2: //Confirm belt is clear
			halt := 0;
			IF (udp_data.state = RunToFront) THEN
				IF rail_mt THEN
					udp_data.state := ReadyToWork;
				END_IF;
			ELSE
				udp_data.state := ReadyToWork;
			END_IF;
	END_CASE;

	// Always clear acknowledgements
	brsmemset(ADR(messages.Read[0]),0,SIZEOF(messages.Read));

END_FUNCTION_BLOCK
```
